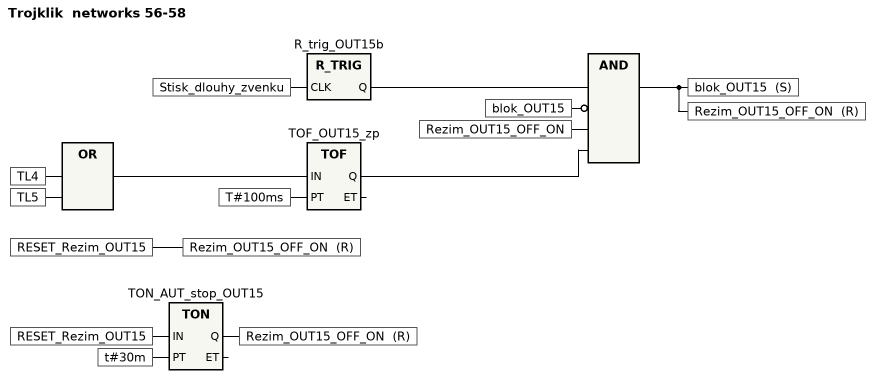
[picture p48: Trojklik (FBD) networks 56-58]
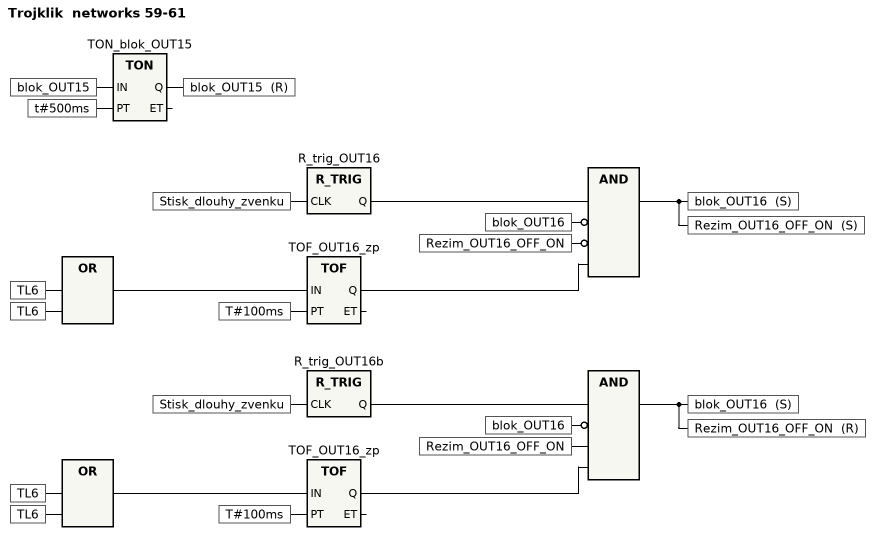
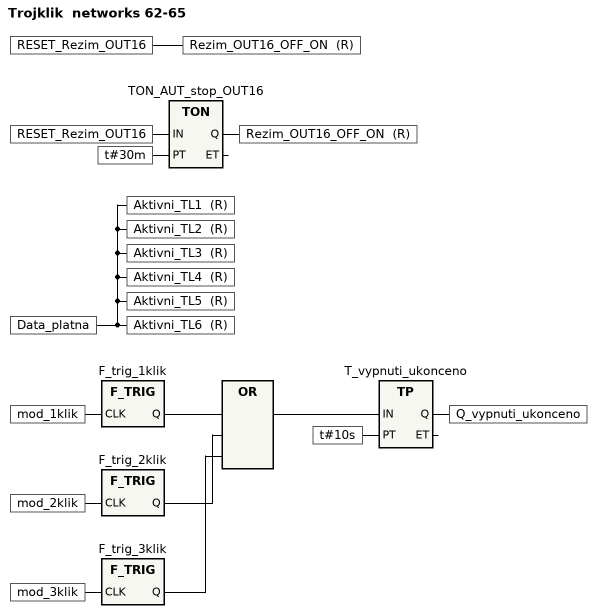
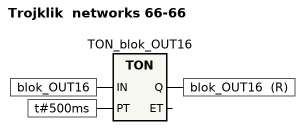
_FBD_ (* Function Block Diagram *)
NETWORK 1
	TP_T_max:TP(IN: T_max:TON(IN: AND(OR(Rezim_1klik_OFF_ON, Rezim_2klik_OFF_ON, Rezim_3klik_OFF_ON), AUT_vyp), PT: cas_vypnuti), PT: t#400ms) => Q_T_MAX
NETWORK 2
	AND(TL1, NOT Aktivni_TL1, NOT Aktivni_TL2, NOT Aktivni_TL3, NOT Aktivni_TL4, NOT Aktivni_TL5, NOT Aktivni_TL6) => S Aktivni_TL1
NETWORK 3
	AND(TL2, NOT Aktivni_TL1, NOT Aktivni_TL2, NOT Aktivni_TL3, NOT Aktivni_TL4, NOT Aktivni_TL5, NOT Aktivni_TL6) => S Aktivni_TL2
NETWORK 4
	AND(TL3, NOT Aktivni_TL1, NOT Aktivni_TL2, NOT Aktivni_TL3, NOT Aktivni_TL4, NOT Aktivni_TL5, NOT Aktivni_TL6) => S Aktivni_TL3
NETWORK 5
	AND(TL4, NOT Aktivni_TL1, NOT Aktivni_TL2, NOT Aktivni_TL3, NOT Aktivni_TL4, NOT Aktivni_TL5, NOT Aktivni_TL6) => S Aktivni_TL4
NETWORK 6
	AND(TL5, NOT Aktivni_TL1, NOT Aktivni_TL2, NOT Aktivni_TL3, NOT Aktivni_TL4, NOT Aktivni_TL5, NOT Aktivni_TL6) => S Aktivni_TL5
NETWORK 7
	AND(TL6, NOT Aktivni_TL1, NOT Aktivni_TL2, NOT Aktivni_TL3, NOT Aktivni_TL4, NOT Aktivni_TL5, NOT Aktivni_TL6) => S Aktivni_TL6
NETWORK 8
	OR(AND(TL1, Aktivni_TL1), AND(TL2, Aktivni_TL2), AND(TL3, Aktivni_TL3)) => TLx_sklad
NETWORK 9
	OR(AND(TL4, Aktivni_TL4), AND(TL5, Aktivni_TL5), AND(TL6, Aktivni_TL6)) => TLx_zvenku
NETWORK 10
	F_trig_hr1:F_TRIG(CLK: TLx_sklad) => TLx_sklad_hr1
NETWORK 11
	F_trig_hr1_zvenku:F_TRIG(CLK: TLx_zvenku) => TLx_sklad_hr1_zvenku
NETWORK 12
	AND(TLx_sklad_hr1, NOT SET_stisk_TLx) => S Stisk_kratky
NETWORK 13
	AND(TLx_sklad_hr1_zvenku, NOT SET_stisk_TLx_zvenku) => S Stisk_kratky_zvenku
NETWORK 14
	TP_byl_kratky:TP(IN: Stisk_kratky, PT: T#4s) => Q_byl_kratky
NETWORK 15
	TP_byl_kratky_zvenku:TP(IN: Stisk_kratky_zvenku, PT: T#4s) => Q_byl_kratky_zvenku
NETWORK 16
	AND(TLx_sklad_hr1, SET_stisk_TLx) => S Stisk_dlouhy
NETWORK 17
	AND(TLx_sklad_hr1_zvenku, SET_stisk_TLx_zvenku) => S Stisk_dlouhy_zvenku
NETWORK 18
	OR(TLx_sklad, TLx_zvenku) => R Stisk_kratky
NETWORK 19
	OR(TLx_zvenku, TLx_sklad) => R Stisk_kratky_zvenku
NETWORK 20
	Stisk_kratky => S blok_kratky
NETWORK 21
	Stisk_kratky_zvenku => S blok_kratky_zvenku
NETWORK 22
	Data_platna => R blok_kratky
NETWORK 23
	Data_platna => R blok_kratky_zvenku
NETWORK 24
	OR(TLx_sklad, TLx_zvenku) => R Stisk_dlouhy
NETWORK 25
	OR(TLx_zvenku, TLx_sklad) => R Stisk_dlouhy_zvenku
NETWORK 26
	AND(NOT mod_1klik, Data_platna, NOT mod_2klik, FALSE, NOT mod_3klik) => R ZAP_VYP_sklad
NETWORK 27
	AND(OR(EQ(TLx_INT, 1), EQ(TLx_INT_zvenku, 1)), NOT mod_1klik, Data_platna, NOT mod_2klik, NOT mod_3klik, NOT ZAP_VYP_sklad, OR(Q_vypnuti_ukonceno, TRUE), NOT blok) => S blok, S mod_1klik
NETWORK 28
	AND(OR(GE(TLx_INT, 1), GE(TLx_INT_zvenku, 1)), OR(Q_vypnuti_ukonceno, TRUE), Data_platna, NOT ZAP_VYP_sklad, NOT blok_ZAP_VYP) => S blok_ZAP_VYP, S ZAP_VYP_sklad
NETWORK 29
	AND(OR(EQ(TLx_INT, 1), EQ(TLx_INT_zvenku, 1)), OR(Data_platna, AND(blok_kratky, TLx_sklad), AND(blok_kratky_zvenku, TLx_zvenku)), ZAP_VYP_sklad, NOT blok_ZAP_VYP, Data_platna, NOT blok_ZAP_VYP, NOT blok) => S blok, R ZAP_VYP_sklad, R mod_1klik
NETWORK 30
	T_blok:TON(IN: blok, PT: T#1s) => R blok
NETWORK 31
	T_blok_ZAP_VYP:TON(IN: blok_ZAP_VYP, PT: T#1s) => R blok_ZAP_VYP
NETWORK 32
	OR(AND(NOT EQ(TLx_INT, 1), NOT EQ(TLx_INT_zvenku, 1), NOT Data_platna, NOT Stisk_dlouhy_zvenku, NOT Stisk_dlouhy, OR(NOT ZAP_VYP_sklad, AND(mod_3klik, FALSE), TRUE, AND(mod_2klik, FALSE)), Data_platna_reset), AND(mod_3klik, FALSE), AND(mod_2klik, FALSE), NOT ZAP_VYP_sklad) => R mod_1klik
NETWORK 33
	AND(OR(EQ(TLx_INT, 2), EQ(TLx_INT_zvenku, 2)), ZAP_VYP_sklad, OR(Q_vypnuti_ukonceno, TRUE), Data_platna) => S mod_2klik
NETWORK 34
	OR(OR(AND(NOT EQ(TLx_INT_zvenku, 2), NOT EQ(TLx_INT, 2), NOT Data_platna, NOT Stisk_dlouhy_zvenku, NOT Stisk_dlouhy, OR(TRUE, NOT ZAP_VYP_sklad, AND(mod_1klik, FALSE), AND(mod_3klik, FALSE)), Data_platna_reset), NOT ZAP_VYP_sklad, AND(mod_3klik, FALSE), AND(mod_1klik, FALSE)), NOT ZAP_VYP_sklad) => R mod_2klik
NETWORK 35
	AND(OR(Q_vypnuti_ukonceno, TRUE), OR(EQ(TLx_INT, 3), EQ(TLx_INT_zvenku, 3)), ZAP_VYP_sklad, Data_platna) => S mod_3klik
NETWORK 36
	OR(OR(AND(NOT EQ(TLx_INT_zvenku, 3), NOT EQ(TLx_INT, 3), NOT Data_platna, NOT Stisk_dlouhy_zvenku, NOT Stisk_dlouhy, OR(TRUE, NOT ZAP_VYP_sklad, AND(mod_1klik, FALSE), AND(mod_2klik, FALSE)), Data_platna_reset), NOT ZAP_VYP_sklad, AND(mod_1klik, FALSE), AND(mod_2klik, FALSE)), NOT ZAP_VYP_sklad) => R mod_3klik
NETWORK 37
	TLx_Citac:CTU(CU: AND(Stisk_kratky, LT(TLx_INT, Pocet_kliku_MAX)), RESET: OR(AND(Data_platna, OR(Q_vypnuti_ukonceno, TRUE)), Q_stisk_TLx), PV: 0, CV => TLx_INT)
NETWORK 38
	TLx_Citac_zvenku:CTU(CU: Stisk_kratky_zvenku, RESET: OR(AND(Data_platna, OR(Q_vypnuti_ukonceno, TRUE)), Q_stisk_TLx_zvenku), PV: 0, CV => TLx_INT_zvenku)
NETWORK 39 (* Data platna *)
	T_Data_platna:TON(IN: AND(NOT TLx_sklad, NOT TLx_zvenku), PT: T#1000ms) => Data_platna
NETWORK 40 (* Data platna *)
	T_Data_platna_reset:TON(IN: AND(NOT TLx_sklad, NOT TLx_zvenku), PT: T#1000ms) => Data_platna_reset
NETWORK 41 (* delka stisku TLx *)
	T_stisk_TLx:TON(IN: AND(TLx_sklad, OR(NOT Q_byl_kratky, TRUE)), PT: T#600ms) => Q_stisk_TLx
NETWORK 42 (* delka stisku TLx *)
	T_stisk_TLx_zvenku:TON(IN: AND(TLx_zvenku, OR(NOT Q_byl_kratky_zvenku, TRUE)), PT: T#600ms) => Q_stisk_TLx_zvenku
NETWORK 43
	SR_stisk_TLx:SR(SET1: Q_stisk_TLx, RESET: R_trig_hr2:R_TRIG(CLK: TLx_sklad)) => SET_stisk_TLx
NETWORK 44
	SR_stisk_TLx_zvenku:SR(SET1: Q_stisk_TLx_zvenku, RESET: R_trig_hr2_zvenku:R_TRIG(CLK: TLx_zvenku)) => SET_stisk_TLx_zvenku
NETWORK 45
	OR(AND(mod_1klik, ZAP_VYP_sklad, TLx_sklad, NOT Q_byl_kratky, mod_1klik, ZAP_VYP_sklad, Q_stisk_TLx), TP_mode_1klik:TP(IN: OR(AND(mod_1klik, ZAP_VYP_sklad, NOT Q_T_MAX, NOT RESET_Rezim_1klik, NOT Q_vypnuti_ukonceno, Data_platna, OR(Stisk_kratky, Stisk_kratky_zvenku)), AND(NOT ZAP_VYP_sklad, OR(Stisk_kratky, Stisk_kratky_zvenku), NOT Q_T_MAX, NOT RESET_Rezim_1klik, FALSE, mod_1klik)), PT: t#400ms), tp_1klik_vyp:TP(IN: AND(f_trig_1klik_vyp:F_TRIG(CLK: mod_1klik), NOT RESET_Rezim_1klik, NOT Q_T_MAX), PT: t#400ms), TP_reset1:TP(IN: AND(mod_1klik, ZAP_VYP_sklad, OR(RESET_Rezim_1klik, Q_T_MAX)), PT: t#400ms)) => Rezim_1klik_PULS
NETWORK 46
	AND(ZAP_VYP_sklad, mod_1klik) => Rezim_1klik_OFF_ON
NETWORK 47
	OR(AND(mod_2klik, ZAP_VYP_sklad, NOT Q_byl_kratky, mod_2klik, ZAP_VYP_sklad, TLx_sklad, Q_stisk_TLx), TP_mode_2klik:TP(IN: OR(AND(mod_2klik, ZAP_VYP_sklad, NOT Q_T_MAX, NOT RESET_Rezim_2klik, NOT Q_vypnuti_ukonceno, Data_platna, OR(Stisk_kratky, Stisk_kratky_zvenku)), AND(NOT ZAP_VYP_sklad, NOT Q_T_MAX, NOT RESET_Rezim_2klik, FALSE, OR(Stisk_kratky, Stisk_kratky_zvenku), mod_2klik)), PT: t#400ms), tp_2klik_vyp:TP(IN: AND(f_trig_2klik_vyp:F_TRIG(CLK: mod_2klik), NOT RESET_Rezim_2klik, NOT Q_T_MAX), PT: t#400ms), TP_reset2:TP(IN: AND(mod_2klik, ZAP_VYP_sklad, OR(RESET_Rezim_2klik, Q_T_MAX)), PT: t#400ms)) => Rezim_2klik_PULS
NETWORK 48
	AND(ZAP_VYP_sklad, mod_2klik) => Rezim_2klik_OFF_ON
NETWORK 49
	OR(AND(mod_3klik, ZAP_VYP_sklad, NOT Q_byl_kratky, mod_3klik, ZAP_VYP_sklad, TLx_sklad, Q_stisk_TLx), TP_mode_3klik:TP(IN: OR(AND(mod_3klik, NOT Q_T_MAX, NOT RESET_Rezim_3klik, NOT Q_vypnuti_ukonceno, Data_platna, ZAP_VYP_sklad, OR(Stisk_kratky, Stisk_kratky_zvenku)), AND(NOT ZAP_VYP_sklad, NOT Q_T_MAX, NOT RESET_Rezim_3klik, FALSE, OR(Stisk_kratky, Stisk_kratky_zvenku), mod_3klik)), PT: t#400ms), tp_3klik_vyp:TP(IN: AND(f_trig_3klik_vyp:F_TRIG(CLK: mod_3klik), NOT RESET_Rezim_3klik, NOT Q_T_MAX), PT: t#400ms), TP_reset3:TP(IN: AND(mod_3klik, ZAP_VYP_sklad, OR(RESET_Rezim_3klik, Q_T_MAX)), PT: t#400ms)) => Rezim_3klik_PULS
NETWORK 50
	AND(ZAP_VYP_sklad, mod_3klik) => Rezim_3klik_OFF_ON
NETWORK 51
	OR(AND(mod_1klik, RESET_Rezim_1klik), AND(mod_2klik, RESET_Rezim_2klik), AND(mod_3klik, RESET_Rezim_3klik), Q_T_MAX) => R ZAP_VYP_sklad
NETWORK 52
	OR(AND(mod_1klik, RESET_Rezim_1klik), Q_T_MAX) => R mod_1klik
NETWORK 53
	OR(AND(mod_2klik, RESET_Rezim_2klik), Q_T_MAX) => R mod_2klik
NETWORK 54
	OR(AND(mod_3klik, RESET_Rezim_3klik), Q_T_MAX) => R mod_3klik
NETWORK 55
	AND(R_trig_OUT15:R_TRIG(CLK: Stisk_dlouhy_zvenku), NOT blok_OUT15, NOT Rezim_OUT15_OFF_ON, TOF_OUT15_zp:TOF(IN: OR(TL4, TL5), PT: T#100ms)) => S blok_OUT15, S Rezim_OUT15_OFF_ON
NETWORK 56
	AND(R_trig_OUT15b:R_TRIG(CLK: Stisk_dlouhy_zvenku), NOT blok_OUT15, Rezim_OUT15_OFF_ON, TOF_OUT15_zp:TOF(IN: OR(TL4, TL5), PT: T#100ms)) => S blok_OUT15, R Rezim_OUT15_OFF_ON
NETWORK 57
	RESET_Rezim_OUT15 => R Rezim_OUT15_OFF_ON
NETWORK 58
	TON_AUT_stop_OUT15:TON(IN: RESET_Rezim_OUT15, PT: t#30m) => R Rezim_OUT15_OFF_ON
NETWORK 59
	TON_blok_OUT15:TON(IN: blok_OUT15, PT: t#500ms) => R blok_OUT15
NETWORK 60
	AND(R_trig_OUT16:R_TRIG(CLK: Stisk_dlouhy_zvenku), NOT blok_OUT16, NOT Rezim_OUT16_OFF_ON, TOF_OUT16_zp:TOF(IN: OR(TL6, TL6), PT: T#100ms)) => S blok_OUT16, S Rezim_OUT16_OFF_ON
NETWORK 61
	AND(R_trig_OUT16b:R_TRIG(CLK: Stisk_dlouhy_zvenku), NOT blok_OUT16, Rezim_OUT16_OFF_ON, TOF_OUT16_zp:TOF(IN: OR(TL6, TL6), PT: T#100ms)) => S blok_OUT16, R Rezim_OUT16_OFF_ON
NETWORK 62
	RESET_Rezim_OUT16 => R Rezim_OUT16_OFF_ON
NETWORK 63
	TON_AUT_stop_OUT16:TON(IN: RESET_Rezim_OUT16, PT: t#30m) => R Rezim_OUT16_OFF_ON
NETWORK 64
	Data_platna => R Aktivni_TL1, R Aktivni_TL2, R Aktivni_TL3, R Aktivni_TL4, R Aktivni_TL5, R Aktivni_TL6
NETWORK 65
	T_vypnuti_ukonceno:TP(IN: OR(F_trig_1klik:F_TRIG(CLK: mod_1klik), F_trig_2klik:F_TRIG(CLK: mod_2klik), F_trig_3klik:F_TRIG(CLK: mod_3klik)), PT: t#10s) => Q_vypnuti_ukonceno
NETWORK 66
	TON_blok_OUT16:TON(IN: blok_OUT16, PT: t#500ms) => R blok_OUT16
_END_FBD_
(* the same logic as Structured Text *)
(* Network 1 *)
T_max(IN := (Rezim_1klik_OFF_ON OR Rezim_2klik_OFF_ON OR Rezim_3klik_OFF_ON) AND AUT_vyp, PT := cas_vypnuti);
TP_T_max(IN := T_max.Q, PT := t#400ms);
Q_T_MAX := TP_T_max.Q;
(* Network 2 *)
IF TL1 AND NOT Aktivni_TL1 AND NOT Aktivni_TL2 AND NOT Aktivni_TL3 AND NOT Aktivni_TL4 AND NOT Aktivni_TL5 AND NOT Aktivni_TL6 THEN Aktivni_TL1 := TRUE; END_IF;
(* Network 3 *)
IF TL2 AND NOT Aktivni_TL1 AND NOT Aktivni_TL2 AND NOT Aktivni_TL3 AND NOT Aktivni_TL4 AND NOT Aktivni_TL5 AND NOT Aktivni_TL6 THEN Aktivni_TL2 := TRUE; END_IF;
(* Network 4 *)
IF TL3 AND NOT Aktivni_TL1 AND NOT Aktivni_TL2 AND NOT Aktivni_TL3 AND NOT Aktivni_TL4 AND NOT Aktivni_TL5 AND NOT Aktivni_TL6 THEN Aktivni_TL3 := TRUE; END_IF;
(* Network 5 *)
IF TL4 AND NOT Aktivni_TL1 AND NOT Aktivni_TL2 AND NOT Aktivni_TL3 AND NOT Aktivni_TL4 AND NOT Aktivni_TL5 AND NOT Aktivni_TL6 THEN Aktivni_TL4 := TRUE; END_IF;
(* Network 6 *)
IF TL5 AND NOT Aktivni_TL1 AND NOT Aktivni_TL2 AND NOT Aktivni_TL3 AND NOT Aktivni_TL4 AND NOT Aktivni_TL5 AND NOT Aktivni_TL6 THEN Aktivni_TL5 := TRUE; END_IF;
(* Network 7 *)
IF TL6 AND NOT Aktivni_TL1 AND NOT Aktivni_TL2 AND NOT Aktivni_TL3 AND NOT Aktivni_TL4 AND NOT Aktivni_TL5 AND NOT Aktivni_TL6 THEN Aktivni_TL6 := TRUE; END_IF;
(* Network 8 *)
TLx_sklad := (TL1 AND Aktivni_TL1) OR (TL2 AND Aktivni_TL2) OR (TL3 AND Aktivni_TL3);
(* Network 9 *)
TLx_zvenku := (TL4 AND Aktivni_TL4) OR (TL5 AND Aktivni_TL5) OR (TL6 AND Aktivni_TL6);
(* Network 10 *)
F_trig_hr1(CLK := TLx_sklad);
TLx_sklad_hr1 := F_trig_hr1.Q;
(* Network 11 *)
F_trig_hr1_zvenku(CLK := TLx_zvenku);
TLx_sklad_hr1_zvenku := F_trig_hr1_zvenku.Q;
(* Network 12 *)
IF TLx_sklad_hr1 AND NOT SET_stisk_TLx THEN Stisk_kratky := TRUE; END_IF;
(* Network 13 *)
IF TLx_sklad_hr1_zvenku AND NOT SET_stisk_TLx_zvenku THEN Stisk_kratky_zvenku := TRUE; END_IF;
(* Network 14 *)
TP_byl_kratky(IN := Stisk_kratky, PT := T#4s);
Q_byl_kratky := TP_byl_kratky.Q;
(* Network 15 *)
TP_byl_kratky_zvenku(IN := Stisk_kratky_zvenku, PT := T#4s);
Q_byl_kratky_zvenku := TP_byl_kratky_zvenku.Q;
(* Network 16 *)
IF TLx_sklad_hr1 AND SET_stisk_TLx THEN Stisk_dlouhy := TRUE; END_IF;
(* Network 17 *)
IF TLx_sklad_hr1_zvenku AND SET_stisk_TLx_zvenku THEN Stisk_dlouhy_zvenku := TRUE; END_IF;
(* Network 18 *)
IF TLx_sklad OR TLx_zvenku THEN Stisk_kratky := FALSE; END_IF;
(* Network 19 *)
IF TLx_zvenku OR TLx_sklad THEN Stisk_kratky_zvenku := FALSE; END_IF;
(* Network 20 *)
IF Stisk_kratky THEN blok_kratky := TRUE; END_IF;
(* Network 21 *)
IF Stisk_kratky_zvenku THEN blok_kratky_zvenku := TRUE; END_IF;
(* Network 22 *)
IF Data_platna THEN blok_kratky := FALSE; END_IF;
(* Network 23 *)
IF Data_platna THEN blok_kratky_zvenku := FALSE; END_IF;
(* Network 24 *)
IF TLx_sklad OR TLx_zvenku THEN Stisk_dlouhy := FALSE; END_IF;
(* Network 25 *)
IF TLx_zvenku OR TLx_sklad THEN Stisk_dlouhy_zvenku := FALSE; END_IF;
(* Network 26 *)
IF NOT mod_1klik AND Data_platna AND NOT mod_2klik AND FALSE AND NOT mod_3klik THEN ZAP_VYP_sklad := FALSE; END_IF;
(* Network 27 *)
_p1 := ((TLx_INT = 1) OR (TLx_INT_zvenku = 1)) AND NOT mod_1klik AND Data_platna AND NOT mod_2klik AND NOT mod_3klik AND NOT ZAP_VYP_sklad AND (Q_vypnuti_ukonceno OR TRUE) AND NOT blok;
IF _p1 THEN blok := TRUE; mod_1klik := TRUE; END_IF;
(* Network 28 *)
_p2 := ((TLx_INT >= 1) OR (TLx_INT_zvenku >= 1)) AND (Q_vypnuti_ukonceno OR TRUE) AND Data_platna AND NOT ZAP_VYP_sklad AND NOT blok_ZAP_VYP;
IF _p2 THEN blok_ZAP_VYP := TRUE; ZAP_VYP_sklad := TRUE; END_IF;
(* Network 29 *)
_p3 := ((TLx_INT = 1) OR (TLx_INT_zvenku = 1)) AND (Data_platna OR (blok_kratky AND TLx_sklad) OR (blok_kratky_zvenku AND TLx_zvenku)) AND ZAP_VYP_sklad AND NOT blok_ZAP_VYP AND Data_platna AND NOT blok_ZAP_VYP AND NOT blok;
IF _p3 THEN blok := TRUE; ZAP_VYP_sklad := FALSE; mod_1klik := FALSE; END_IF;
(* Network 30 *)
T_blok(IN := blok, PT := T#1s);
IF T_blok.Q THEN blok := FALSE; END_IF;
(* Network 31 *)
T_blok_ZAP_VYP(IN := blok_ZAP_VYP, PT := T#1s);
IF T_blok_ZAP_VYP.Q THEN blok_ZAP_VYP := FALSE; END_IF;
(* Network 32 *)
IF (NOT (TLx_INT = 1) AND NOT (TLx_INT_zvenku = 1) AND NOT Data_platna AND NOT Stisk_dlouhy_zvenku AND NOT Stisk_dlouhy AND (NOT ZAP_VYP_sklad OR (mod_3klik AND FALSE) OR TRUE OR (mod_2klik AND FALSE)) AND Data_platna_reset) OR (mod_3klik AND FALSE) OR (mod_2klik AND FALSE) OR NOT ZAP_VYP_sklad THEN mod_1klik := FALSE; END_IF;
(* Network 33 *)
IF ((TLx_INT = 2) OR (TLx_INT_zvenku = 2)) AND ZAP_VYP_sklad AND (Q_vypnuti_ukonceno OR TRUE) AND Data_platna THEN mod_2klik := TRUE; END_IF;
(* Network 34 *)
IF ((NOT (TLx_INT_zvenku = 2) AND NOT (TLx_INT = 2) AND NOT Data_platna AND NOT Stisk_dlouhy_zvenku AND NOT Stisk_dlouhy AND (TRUE OR NOT ZAP_VYP_sklad OR (mod_1klik AND FALSE) OR (mod_3klik AND FALSE)) AND Data_platna_reset) OR NOT ZAP_VYP_sklad OR (mod_3klik AND FALSE) OR (mod_1klik AND FALSE)) OR NOT ZAP_VYP_sklad THEN mod_2klik := FALSE; END_IF;
(* Network 35 *)
IF (Q_vypnuti_ukonceno OR TRUE) AND ((TLx_INT = 3) OR (TLx_INT_zvenku = 3)) AND ZAP_VYP_sklad AND Data_platna THEN mod_3klik := TRUE; END_IF;
(* Network 36 *)
IF ((NOT (TLx_INT_zvenku = 3) AND NOT (TLx_INT = 3) AND NOT Data_platna AND NOT Stisk_dlouhy_zvenku AND NOT Stisk_dlouhy AND (TRUE OR NOT ZAP_VYP_sklad OR (mod_1klik AND FALSE) OR (mod_2klik AND FALSE)) AND Data_platna_reset) OR NOT ZAP_VYP_sklad OR (mod_1klik AND FALSE) OR (mod_2klik AND FALSE)) OR NOT ZAP_VYP_sklad THEN mod_3klik := FALSE; END_IF;
(* Network 37 *)
TLx_Citac(CU := Stisk_kratky AND (TLx_INT < Pocet_kliku_MAX), RESET := (Data_platna AND (Q_vypnuti_ukonceno OR TRUE)) OR Q_stisk_TLx, PV := 0);
TLx_INT := TLx_Citac.CV;
(* Network 38 *)
TLx_Citac_zvenku(CU := Stisk_kratky_zvenku, RESET := (Data_platna AND (Q_vypnuti_ukonceno OR TRUE)) OR Q_stisk_TLx_zvenku, PV := 0);
TLx_INT_zvenku := TLx_Citac_zvenku.CV;
(* Network 39 *)
T_Data_platna(IN := NOT TLx_sklad AND NOT TLx_zvenku, PT := T#1000ms);
Data_platna := T_Data_platna.Q;
(* Network 40 *)
T_Data_platna_reset(IN := NOT TLx_sklad AND NOT TLx_zvenku, PT := T#1000ms);
Data_platna_reset := T_Data_platna_reset.Q;
(* Network 41: see the listing above *)
(* Network 42: see the listing above *)
(* Network 43 *)
R_trig_hr2(CLK := TLx_sklad);
SR_stisk_TLx(SET1 := Q_stisk_TLx, RESET := R_trig_hr2.Q);
SET_stisk_TLx := SR_stisk_TLx.Q1;
(* Network 44 *)
R_trig_hr2_zvenku(CLK := TLx_zvenku);
SR_stisk_TLx_zvenku(SET1 := Q_stisk_TLx_zvenku, RESET := R_trig_hr2_zvenku.Q);
SET_stisk_TLx_zvenku := SR_stisk_TLx_zvenku.Q1;
(* Network 45 *)
TP_mode_1klik(IN := (mod_1klik AND ZAP_VYP_sklad AND NOT Q_T_MAX AND NOT RESET_Rezim_1klik AND NOT Q_vypnuti_ukonceno AND Data_platna AND (Stisk_kratky OR Stisk_kratky_zvenku)) OR (NOT ZAP_VYP_sklad AND (Stisk_kratky OR Stisk_kratky_zvenku) AND NOT Q_T_MAX AND NOT RESET_Rezim_1klik AND FALSE AND mod_1klik), PT := t#400ms);
f_trig_1klik_vyp(CLK := mod_1klik);
tp_1klik_vyp(IN := f_trig_1klik_vyp.Q AND NOT RESET_Rezim_1klik AND NOT Q_T_MAX, PT := t#400ms);
TP_reset1(IN := mod_1klik AND ZAP_VYP_sklad AND (RESET_Rezim_1klik OR Q_T_MAX), PT := t#400ms);
Rezim_1klik_PULS := (mod_1klik AND ZAP_VYP_sklad AND TLx_sklad AND NOT Q_byl_kratky AND mod_1klik AND ZAP_VYP_sklad AND Q_stisk_TLx) OR TP_mode_1klik.Q OR tp_1klik_vyp.Q OR TP_reset1.Q;
(* Network 46 *)
Rezim_1klik_OFF_ON := ZAP_VYP_sklad AND mod_1klik;
(* Network 47 *)
TP_mode_2klik(IN := (mod_2klik AND ZAP_VYP_sklad AND NOT Q_T_MAX AND NOT RESET_Rezim_2klik AND NOT Q_vypnuti_ukonceno AND Data_platna AND (Stisk_kratky OR Stisk_kratky_zvenku)) OR (NOT ZAP_VYP_sklad AND NOT Q_T_MAX AND NOT RESET_Rezim_2klik AND FALSE AND (Stisk_kratky OR Stisk_kratky_zvenku) AND mod_2klik), PT := t#400ms);
f_trig_2klik_vyp(CLK := mod_2klik);
tp_2klik_vyp(IN := f_trig_2klik_vyp.Q AND NOT RESET_Rezim_2klik AND NOT Q_T_MAX, PT := t#400ms);
TP_reset2(IN := mod_2klik AND ZAP_VYP_sklad AND (RESET_Rezim_2klik OR Q_T_MAX), PT := t#400ms);
Rezim_2klik_PULS := (mod_2klik AND ZAP_VYP_sklad AND NOT Q_byl_kratky AND mod_2klik AND ZAP_VYP_sklad AND TLx_sklad AND Q_stisk_TLx) OR TP_mode_2klik.Q OR tp_2klik_vyp.Q OR TP_reset2.Q;
(* Network 48 *)
Rezim_2klik_OFF_ON := ZAP_VYP_sklad AND mod_2klik;
(* Network 49 *)
TP_mode_3klik(IN := (mod_3klik AND NOT Q_T_MAX AND NOT RESET_Rezim_3klik AND NOT Q_vypnuti_ukonceno AND Data_platna AND ZAP_VYP_sklad AND (Stisk_kratky OR Stisk_kratky_zvenku)) OR (NOT ZAP_VYP_sklad AND NOT Q_T_MAX AND NOT RESET_Rezim_3klik AND FALSE AND (Stisk_kratky OR Stisk_kratky_zvenku) AND mod_3klik), PT := t#400ms);
f_trig_3klik_vyp(CLK := mod_3klik);
tp_3klik_vyp(IN := f_trig_3klik_vyp.Q AND NOT RESET_Rezim_3klik AND NOT Q_T_MAX, PT := t#400ms);
TP_reset3(IN := mod_3klik AND ZAP_VYP_sklad AND (RESET_Rezim_3klik OR Q_T_MAX), PT := t#400ms);
Rezim_3klik_PULS := (mod_3klik AND ZAP_VYP_sklad AND NOT Q_byl_kratky AND mod_3klik AND ZAP_VYP_sklad AND TLx_sklad AND Q_stisk_TLx) OR TP_mode_3klik.Q OR tp_3klik_vyp.Q OR TP_reset3.Q;
(* Network 50 *)
Rezim_3klik_OFF_ON := ZAP_VYP_sklad AND mod_3klik;
(* Network 51 *)
IF (mod_1klik AND RESET_Rezim_1klik) OR (mod_2klik AND RESET_Rezim_2klik) OR (mod_3klik AND RESET_Rezim_3klik) OR Q_T_MAX THEN ZAP_VYP_sklad := FALSE; END_IF;
(* Network 52 *)
IF (mod_1klik AND RESET_Rezim_1klik) OR Q_T_MAX THEN mod_1klik := FALSE; END_IF;
(* Network 53 *)
IF (mod_2klik AND RESET_Rezim_2klik) OR Q_T_MAX THEN mod_2klik := FALSE; END_IF;
(* Network 54 *)
IF (mod_3klik AND RESET_Rezim_3klik) OR Q_T_MAX THEN mod_3klik := FALSE; END_IF;
(* Network 55 *)
R_trig_OUT15(CLK := Stisk_dlouhy_zvenku);
TOF_OUT15_zp(IN := TL4 OR TL5, PT := T#100ms);
_p4 := R_trig_OUT15.Q AND NOT blok_OUT15 AND NOT Rezim_OUT15_OFF_ON AND TOF_OUT15_zp.Q;
IF _p4 THEN blok_OUT15 := TRUE; Rezim_OUT15_OFF_ON := TRUE; END_IF;
(* Network 56 *)
R_trig_OUT15b(CLK := Stisk_dlouhy_zvenku);
TOF_OUT15_zp(IN := TL4 OR TL5, PT := T#100ms);
_p5 := R_trig_OUT15b.Q AND NOT blok_OUT15 AND Rezim_OUT15_OFF_ON AND TOF_OUT15_zp.Q;
IF _p5 THEN blok_OUT15 := TRUE; Rezim_OUT15_OFF_ON := FALSE; END_IF;
(* Network 57 *)
IF RESET_Rezim_OUT15 THEN Rezim_OUT15_OFF_ON := FALSE; END_IF;
(* Network 58 *)
TON_AUT_stop_OUT15(IN := RESET_Rezim_OUT15, PT := t#30m);
IF TON_AUT_stop_OUT15.Q THEN Rezim_OUT15_OFF_ON := FALSE; END_IF;
(* Network 59 *)
TON_blok_OUT15(IN := blok_OUT15, PT := t#500ms);
IF TON_blok_OUT15.Q THEN blok_OUT15 := FALSE; END_IF;
(* Network 60 *)
R_trig_OUT16(CLK := Stisk_dlouhy_zvenku);
TOF_OUT16_zp(IN := TL6 OR TL6, PT := T#100ms);
_p6 := R_trig_OUT16.Q AND NOT blok_OUT16 AND NOT Rezim_OUT16_OFF_ON AND TOF_OUT16_zp.Q;
IF _p6 THEN blok_OUT16 := TRUE; Rezim_OUT16_OFF_ON := TRUE; END_IF;
(* Network 61 *)
R_trig_OUT16b(CLK := Stisk_dlouhy_zvenku);
TOF_OUT16_zp(IN := TL6 OR TL6, PT := T#100ms);
_p7 := R_trig_OUT16b.Q AND NOT blok_OUT16 AND Rezim_OUT16_OFF_ON AND TOF_OUT16_zp.Q;
IF _p7 THEN blok_OUT16 := TRUE; Rezim_OUT16_OFF_ON := FALSE; END_IF;
(* Network 62 *)
IF RESET_Rezim_OUT16 THEN Rezim_OUT16_OFF_ON := FALSE; END_IF;
(* Network 63 *)
TON_AUT_stop_OUT16(IN := RESET_Rezim_OUT16, PT := t#30m);
IF TON_AUT_stop_OUT16.Q THEN Rezim_OUT16_OFF_ON := FALSE; END_IF;
(* Network 64 *)
IF Data_platna THEN Aktivni_TL1 := FALSE; Aktivni_TL2 := FALSE; Aktivni_TL3 := FALSE; Aktivni_TL4 := FALSE; Aktivni_TL5 := FALSE; Aktivni_TL6 := FALSE; END_IF;
(* Network 65 *)
F_trig_1klik(CLK := mod_1klik);
F_trig_2klik(CLK := mod_2klik);
F_trig_3klik(CLK := mod_3klik);
T_vypnuti_ukonceno(IN := F_trig_1klik.Q OR F_trig_2klik.Q OR F_trig_3klik.Q, PT := t#10s);
Q_vypnuti_ukonceno := T_vypnuti_ukonceno.Q;
(* Network 66 *)
TON_blok_OUT16(IN := blok_OUT16, PT := t#500ms);
IF TON_blok_OUT16.Q THEN blok_OUT16 := FALSE; END_IF;
END_FUNCTION_BLOCK

(* POU Zhasni, ST *)
FUNCTION_BLOCK Zhasni
VAR_INPUT
	wIn: WORD;
	xPresun: BOOL;
END_VAR
VAR_OUTPUT
	xonOUT1: BOOL;
	xonOUT2: BOOL;
	xonOUT3: BOOL;

	xoffOUT1: BOOL;
	xoffOUT2: BOOL;
	xoffOUT3: BOOL;
	wLast: WORD;
	xPresunuto: BOOL;
END_VAR
VAR
	start: BOOL;
	TP1: TP;
	stav: WORD;
	last: WORD;
	F_TRIG5: F_TRIG;
END_VAR
IF xPresun=TRUE THEN
	stav:=wIn;
	start:=TRUE;


CASE stav OF
	2: 	xonOUT2:=TRUE;
		last:=2;
	3: 	xonOUT3:=TRUE;
		last:=3;
END_CASE


IF wLast=0 AND stav=1 THEN
xonOUT1:=TRUE;
last:=1;
END_IF

IF NOT( wLast=0) AND stav=1 THEN
	CASE wLast OF
	1: xoffOUT1:=TRUE;
		last:=0;
	2: xoffOUT2:=TRUE;
		last:=0;
	3: xoffOUT3:=TRUE;
		last:=0;
	END_CASE

END_IF
END_IF

TP1(IN:=start , PT:=t#50ms , Q=> , ET=> );
F_TRIG5(CLK:=TP1.Q , Q=> );
IF F_TRIG5.Q=TRUE THEN
	wLast:=last;
	start:=FALSE;
	xoffOUT1:=FALSE;
	xoffOUT2:=FALSE;
	xoffOUT3:=FALSE;
	xonOUT1:=FALSE;
	xonOUT2:=FALSE;
	xonOUT3:=FALSE;
END_IF

xPresunuto:=xPresun;
END_FUNCTION_BLOCK

(* POU dali/Ovladani_7_8_9, ST *)
FUNCTION_BLOCK Ovladani_7_8_9
VAR_INPUT
	xVstup: BOOL;
	rCidlo: REAL;
	rUroven1: REAL;
	rUroven2: REAL;
	tZpozdeniCidla: TIME;
END_VAR
VAR_OUTPUT
	On_7: BOOL;
	On_8: BOOL;
	On_9: BOOL;
	Off_7: BOOL;
	Off_8: BOOL;
	Off_9: BOOL;
END_VAR
VAR
	Stav7: BOOL;
	Stav8: BOOL;
	Stav9: BOOL;
	StavSvetel: BOOL;
	Zmacknuto: BOOL;
	R_TRIG1: R_TRIG;
	F_TRIG1: F_TRIG;
	BLINK1: BLINK;

END_VAR
R_TRIG1(CLK:=xVstup, Q=>Zmacknuto );
F_TRIG1(CLK:=xVstup);
BLINK1(ENABLE:=TRUE , TIMELOW:=tZpozdeniCidla , TIMEHIGH:=t#1s);

IF BLINK1.OUT THEN Cidlo_zpozdene:=rCidlo;
END_IF

StavSvetel:=Stav7 OR Stav8 OR Stav9;

IF Zmacknuto AND (StavSvetel=FALSE) THEN		(*vse zhasnuto*)
	On_7:=TRUE;
	On_8:=TRUE;
	On_9:=TRUE;
	Stav7:=TRUE;
	Stav8:=TRUE;
	Stav9:=TRUE;
END_IF

IF Zmacknuto AND (StavSvetel=TRUE) THEN		(*neco rozsviceno*)
	Off_7:=TRUE;
	Off_8:=TRUE;
	Off_9:=TRUE;
	Stav7:=FALSE;
	Stav8:=FALSE;
	Stav9:=FALSE;
END_IF

IF F_TRIG1.Q THEN
	On_7:=FALSE;
	On_8:=FALSE;
	On_9:=FALSE;
	Off_7:=FALSE;
	Off_8:=FALSE;
	Off_9:=FALSE;
END_IF

IF Cidlo_zpozdene>rUroven1 THEN
	On_7:=FALSE;
	Off_7:=TRUE;
	Stav7:=FALSE;
ELSIF StavSvetel THEN
	On_7:=TRUE;
	Off_7:=FALSE;
	Stav7:=TRUE;
END_IF

IF Cidlo_zpozdene>rUroven2 THEN
	On_9:=FALSE;
	Off_9:=TRUE;
	Stav9:=FALSE;
ELSIF StavSvetel THEN
	On_9:=TRUE;
	Off_9:=FALSE;
	Stav9:=TRUE;
END_IF

IF Zmacknuto AND (StavSvetel=TRUE) THEN		(*neco rozsviceno*)
	Off_7:=TRUE;
	Off_8:=TRUE;
	Off_9:=TRUE;
	Stav7:=FALSE;
	Stav8:=FALSE;
	Stav9:=FALSE;
END_IF

IF F_TRIG1.Q THEN
	On_7:=FALSE;
	On_8:=FALSE;
	On_9:=FALSE;
	Off_7:=FALSE;
	Off_8:=FALSE;
	Off_9:=FALSE;
END_IF
END_FUNCTION_BLOCK

(* POU TriFaze, ST *)
PROGRAM TriFaze
VAR

	Fb750_493_Master3Phase1: Fb750_493_Master3Phase;
	abIn AT %IB22: ARRAY [0..11] OF BYTE;
	abOut AT %QB6: ARRAY [0..11] OF BYTE;

	typ3faze: typConfig3Phase;
	awProud: ARRAY [1..3] OF WORD;
	awNapeti: ARRAY [1..3] OF WORD;
	aiCosFi: ARRAY [1..3] OF INT;
	aiVykon: ARRAY [1..3] OF INT;
	adwSpotreba: ARRAY [1..3] OF DWORD;

	arProud: ARRAY [1..3] OF REAL;
	arNapeti: ARRAY [1..3] OF REAL;
	arCosFi: ARRAY [1..3] OF REAL;
	arVykon: ARRAY [1..3] OF REAL;
	arSpotreba: ARRAY [1..3] OF REAL;
	SmazL1: BOOL;
	SmazL2: BOOL;
	SmazL3: BOOL;
END_VAR
Fb750_493_Master3Phase1(
	xEnable:= TRUE,
	tCycleTime:= ,
	x750_493_000_001:=FALSE ,
	xSaveEnergyConsumption:= ,
	xDeleteEnergyConsumptionL1:=SmazL1 ,
	xDeleteEnergyConsumptionL2:=SmazL1 ,
	xDeleteEnergyConsumptionL3:=SmazL1 ,
	abIn_Data_750_493:=abIn ,
	abOut_Data_750_493:=abOut ,
	typConfig3Phase:=typ3faze ,
	xReady=> ,
	abError=> , 
	awCurrent=>awProud ,
	awVoltage=>awNapeti ,
	aiPowerFactor=>aiCosFi ,
	aiEffectivePower=>aiVykon ,
	adwEnergyConsumption=>adwSpotreba ,
	awMaxCurrent=> , 
	awMaxVoltage=> , 
	awMinCurrent=> ,
	awMinVoltage=> );

arProud[1]:=awProud[1]/1000.0;
arProud[2]:=awProud[2]/1000.0;
arProud[3]:=awProud[3]/1000.0;

arNapeti[1]:=awNapeti[1]/10.0;
arNapeti[2]:=awNapeti[2]/10.0;
arNapeti[3]:=awNapeti[3]/10.0;

arCosFi[1]:=aiCosFi[1]/100.0;
arCosFi[2]:=aiCosFi[2]/100.0;
arCosFi[3]:=aiCosFi[3]/100.0;

arVykon[1]:=aiVykon[1]/10000.0;
arVykon[2]:=aiVykon[2]/10000.0;
arVykon[3]:=aiVykon[3]/10000.0;
;
END_PROGRAM

(* POU PrirazeniVzdalenychPromenych, CFC *)
PROGRAM PrirazeniVzdalenychPromenych
VAR
	d1: D_klop;
	d2: D_klop;
	d3: D_klop;
	d4: D_klop;
	d5: D_klop;
	d6: D_klop;
	d7: D_klop;
	d8: D_klop;
END_VAR
VAR (* helpers for the ST form of the networks *)
	_t91 : REAL;
END_VAR
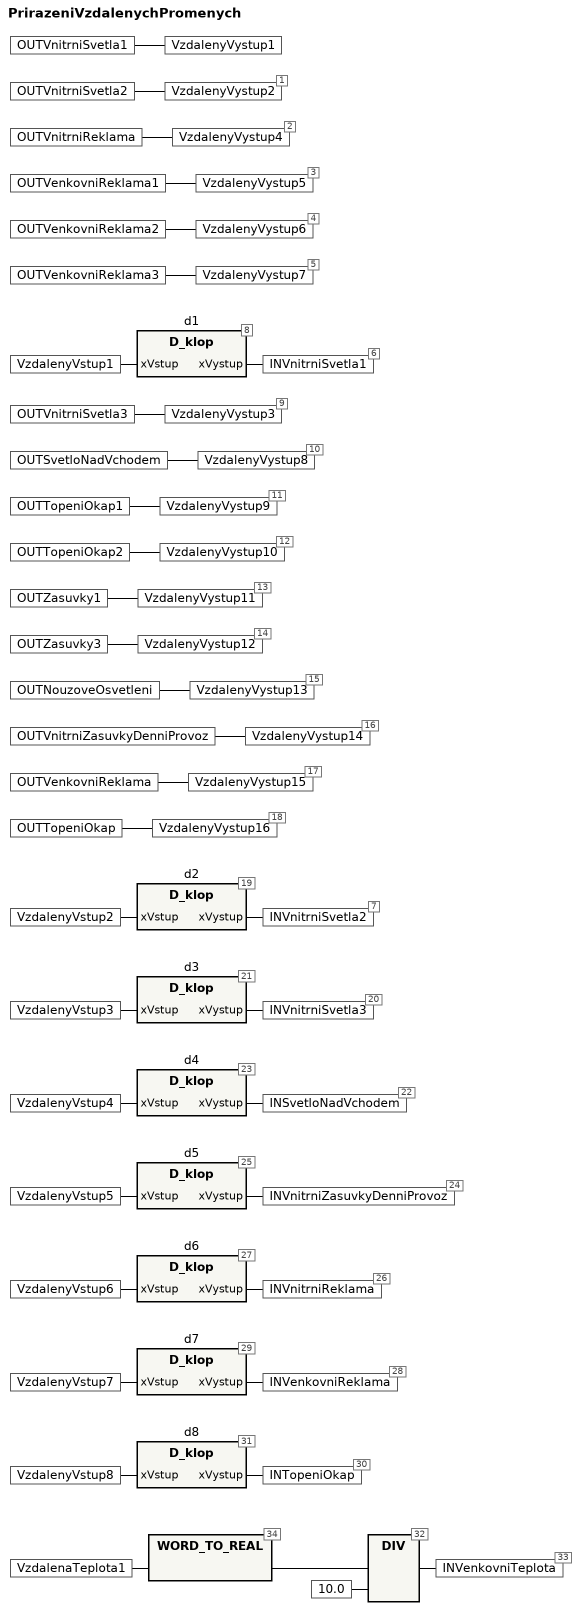
_CFC_ (* Continuous Function Chart, elements in execution order *)
#0 VzdalenyVystup1 <= OUTVnitrniSvetla1
#1 VzdalenyVystup2 <= OUTVnitrniSvetla2
#2 VzdalenyVystup4 <= OUTVnitrniReklama
#3 VzdalenyVystup5 <= OUTVenkovniReklama1
#4 VzdalenyVystup6 <= OUTVenkovniReklama2
#5 VzdalenyVystup7 <= OUTVenkovniReklama3
#6 INVnitrniSvetla1 <= #8.xVystup
#7 INVnitrniSvetla2 <= #19.xVystup
#8 d1:D_klop(xVstup: VzdalenyVstup1)
#9 VzdalenyVystup3 <= OUTVnitrniSvetla3
#10 VzdalenyVystup8 <= OUTSvetloNadVchodem
#11 VzdalenyVystup9 <= OUTTopeniOkap1
#12 VzdalenyVystup10 <= OUTTopeniOkap2
#13 VzdalenyVystup11 <= OUTZasuvky1
#14 VzdalenyVystup12 <= OUTZasuvky3
#15 VzdalenyVystup13 <= OUTNouzoveOsvetleni
#16 VzdalenyVystup14 <= OUTVnitrniZasuvkyDenniProvoz
#17 VzdalenyVystup15 <= OUTVenkovniReklama
#18 VzdalenyVystup16 <= OUTTopeniOkap
#19 d2:D_klop(xVstup: VzdalenyVstup2)
#20 INVnitrniSvetla3 <= #21.xVystup
#21 d3:D_klop(xVstup: VzdalenyVstup3)
#22 INSvetloNadVchodem <= #23.xVystup
#23 d4:D_klop(xVstup: VzdalenyVstup4)
#24 INVnitrniZasuvkyDenniProvoz <= #25.xVystup
#25 d5:D_klop(xVstup: VzdalenyVstup5)
#26 INVnitrniReklama <= #27.xVystup
#27 d6:D_klop(xVstup: VzdalenyVstup6)
#28 INVenkovniReklama <= #29.xVystup
#29 d7:D_klop(xVstup: VzdalenyVstup7)
#30 INTopeniOkap <= #31.xVystup
#31 d8:D_klop(xVstup: VzdalenyVstup8)
#32 DIV(#34, 10.0)
#33 INVenkovniTeplota <= #32
#34 WORD_TO_REAL(VzdalenaTeplota1)
_END_CFC_
(* the same logic as Structured Text *)
VzdalenyVystup1 := OUTVnitrniSvetla1;
VzdalenyVystup2 := OUTVnitrniSvetla2;
VzdalenyVystup4 := OUTVnitrniReklama;
VzdalenyVystup5 := OUTVenkovniReklama1;
VzdalenyVystup6 := OUTVenkovniReklama2;
VzdalenyVystup7 := OUTVenkovniReklama3;
INVnitrniSvetla1 := d1.xVystup;
INVnitrniSvetla2 := d2.xVystup;
d1(xVstup := VzdalenyVstup1);
VzdalenyVystup3 := OUTVnitrniSvetla3;
VzdalenyVystup8 := OUTSvetloNadVchodem;
VzdalenyVystup9 := OUTTopeniOkap1;
VzdalenyVystup10 := OUTTopeniOkap2;
VzdalenyVystup11 := OUTZasuvky1;
VzdalenyVystup12 := OUTZasuvky3;
VzdalenyVystup13 := OUTNouzoveOsvetleni;
VzdalenyVystup14 := OUTVnitrniZasuvkyDenniProvoz;
VzdalenyVystup15 := OUTVenkovniReklama;
VzdalenyVystup16 := OUTTopeniOkap;
d2(xVstup := VzdalenyVstup2);
INVnitrniSvetla3 := d3.xVystup;
d3(xVstup := VzdalenyVstup3);
INSvetloNadVchodem := d4.xVystup;
d4(xVstup := VzdalenyVstup4);
INVnitrniZasuvkyDenniProvoz := d5.xVystup;
d5(xVstup := VzdalenyVstup5);
INVnitrniReklama := d6.xVystup;
d6(xVstup := VzdalenyVstup6);
INVenkovniReklama := d7.xVystup;
d7(xVstup := VzdalenyVstup7);
INTopeniOkap := d8.xVystup;
d8(xVstup := VzdalenyVstup8);
INVenkovniTeplota := _t91 / 10.0;
_t91 := WORD_TO_REAL(VzdalenaTeplota1);
END_PROGRAM

(* POU Ostatni/D_klop, ST *)
FUNCTION_BLOCK D_klop
VAR_INPUT
	xVstup: BOOL;
END_VAR
VAR_OUTPUT
	xVystup: BOOL;
END_VAR
VAR
	p: BOOL:= FALSE;
	a: BOOL:= TRUE;
END_VAR
IF(xVstup)
THEN
	IF(p)
	THEN
		IF (a)
			THEN
			xVystup := FALSE;
			p := FALSE;
			a := FALSE;
		END_IF
	ELSE
		IF (a)
			THEN
			xVystup := TRUE;
			p := TRUE;
			a := FALSE;
		END_IF
	END_IF
ELSE
	a:= TRUE;
END_IF
END_FUNCTION_BLOCK

(* POU ProdejnaMaterialu, FBD *)
PROGRAM ProdejnaMaterialu
VAR
	NEVIM: BOOL;
	zasuvky: IntervalSepnuti;
	PRGVnitrniZasuvkyDenniProvoz: BOOL;
	iZasuvkyStartHodiny: INT := 17;
	iZasuvkyStartMinuty: INT := 0;
	iZasuvkyKonecHodiny: INT := 6;
	iZasuvkyKonecMinuty: INT := 0;

	SvetloNadVchodem1: IntervalSepnuti;
	PRGSvetloNadVchodem: BOOL;
	iSvetloNadVchodemStartHodiny1: INT:= 8;
	iSvetloNadVchodemStartMinuty1: INT:= 0;
	iSvetloNadVchodemKonecHodiny1: INT:= 17;
	iSvetloNadVchodemKonecMinuty1: INT:= 0;
	rUrovenSvetlonadVchodem1: REAL;
	SvetloNadVchodem2: IntervalSepnuti;
	iSvetloNadVchodemStartHodiny2: INT:= 8;
	iSvetloNadVchodemStartMinuty2: INT:= 0;
	iSvetloNadVchodemKonecHodiny2: INT:= 17;
	iSvetloNadVchodemKonecMinuty2: INT:= 0;
	rUrovenSvetlonadVchodem2: REAL;
	xSvetloNadVchodemPracTyden: BOOL;
	xSvetloNadVchodemVikend: BOOL;

	iVnitrniReklamaStartHodiny1: INT:= 17;
	iVnitrniReklamaStartMinuty1: INT:= 0;
	iVnitrniReklamaKonecHodiny1: INT:= 22;
	iVnitrniReklamakonecMinuty1: INT:= 0;
	iVnitrniReklamaStartHodiny2: INT:= 5;
	iVnitrniReklamaStartMinuty2: INT:= 30;
	iVnitrniReklamaKonecHodiny2: INT:= 8;
	iVnitrniReklamakonecMinuty2: INT:= 0;
	NocniRezimVnitrniReklama1: IntervalSepnuti;
	NocniRezimVnitrniReklama2: IntervalSepnuti;
	PRGVnitrniReklama: BOOL;

	TeplotaVenkovniMAX: REAL:= 5.0;
	TeplotaVenkovniMIN: REAL:= -5.0;

	VnitrniSvetla1: IntervalSepnuti;
	VnitrniSvetla2: IntervalSepnuti;
	PRGVnitrniSvetla1: BOOL;
	iVnitrniSvetlaStartHodiny1: INT:= 6;
	iVnitrniSvetlaStartMinuty1: INT:= 45;
	iVnitrniSvetlaKonecHodiny1: INT:= 18;
	iVnitrniSvetlaKonecMinuty1: INT:= 0;
	rIntenzitaVnitrniSvetla1 : INT;
	iVnitrniSvetlaStartHodiny2: INT:= 6;
	iVnitrniSvetlaStartMinuty2: INT:= 45;
	iVnitrniSvetlaKonecHodiny2: INT:= 18;
	iVnitrniSvetlaKonecMinuty2: INT:= 0;
	rIntenzitaVnitrniSvetla2 : INT;
	xVnitrniSvetla1PracDen: BOOL;
	xVnitrniSvetla1Vikend: BOOL;

	VnitrniSvetla3: IntervalSepnuti;
	VnitrniSvetla4: IntervalSepnuti;
	PRGVnitrniSvetla2: BOOL;
	iVnitrniSvetlaStartHodiny3: INT:= 6;
	iVnitrniSvetlaStartMinuty3: INT:= 45;
	iVnitrniSvetlaKonecHodiny3: INT:= 18;
	iVnitrniSvetlaKonecMinuty3: INT:= 0;
	rIntenzitaVnitrniSvetla3 : INT;
	iVnitrniSvetlaStartHodiny4: INT:= 6;
	iVnitrniSvetlaStartMinuty4: INT:= 45;
	iVnitrniSvetlaKonecHodiny4: INT:= 18;
	iVnitrniSvetlaKonecMinuty4: INT:= 0;
	rIntenzitaVnitrniSvetla4 : INT;
	xVnitrniSvetla2PracDen: BOOL;
	xVnitrniSvetla2Vikend: BOOL;

	VnitrniSvetla5: IntervalSepnuti;
	VnitrniSvetla6: IntervalSepnuti;
	PRGVnitrniSvetla3: BOOL;
	iVnitrniSvetlaStartHodiny5: INT:= 6;
	iVnitrniSvetlaStartMinuty5: INT:= 45;
	iVnitrniSvetlaKonecHodiny5: INT:= 18;
	iVnitrniSvetlaKonecMinuty5: INT:= 0;
	rIntenzitaVnitrniSvetla5 : INT;
	iVnitrniSvetlaStartHodiny6: INT:= 6;
	iVnitrniSvetlaStartMinuty6: INT:= 45;
	iVnitrniSvetlaKonecHodiny6: INT:= 18;
	iVnitrniSvetlaKonecMinuty6: INT:= 0;
	rIntenzitaVnitrniSvetla6 : INT;
	xVnitrniSvetla3PracDen: BOOL;
	xVnitrniSvetla3Vikend: BOOL;
END_VAR
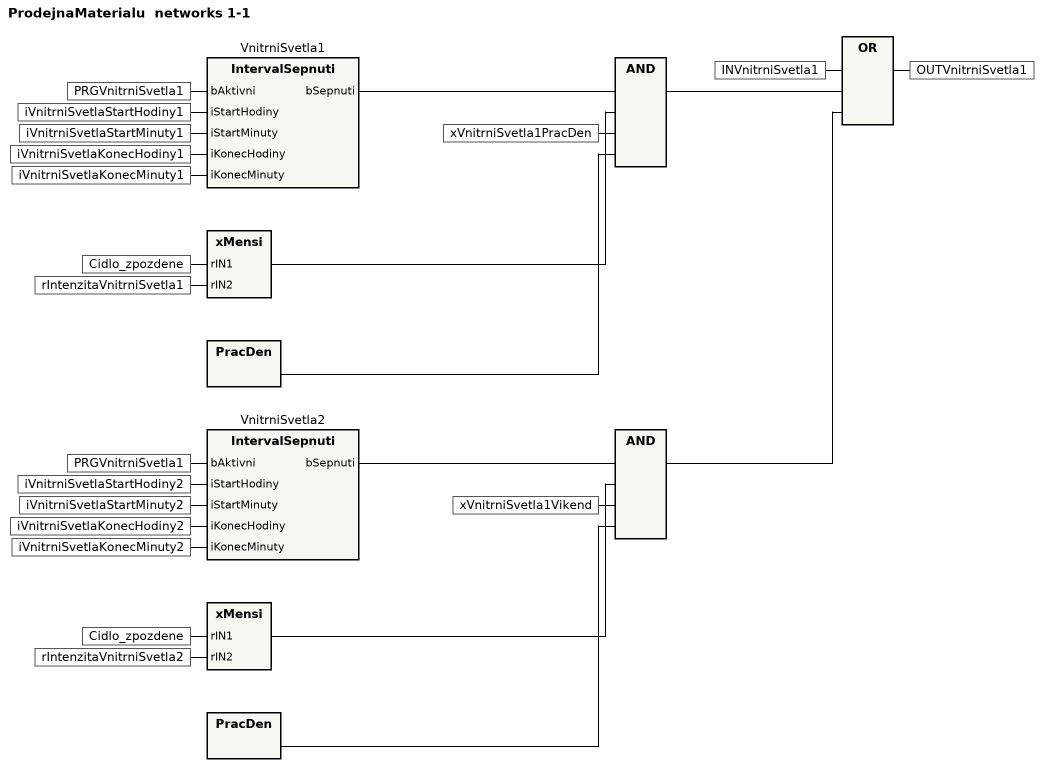
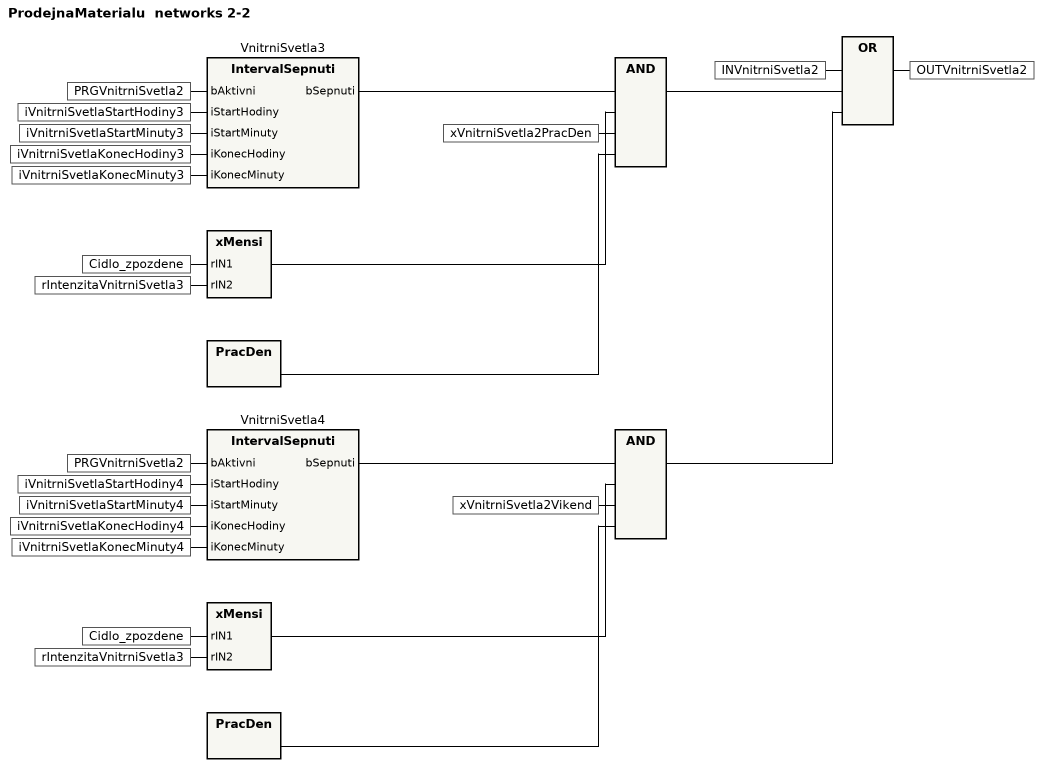
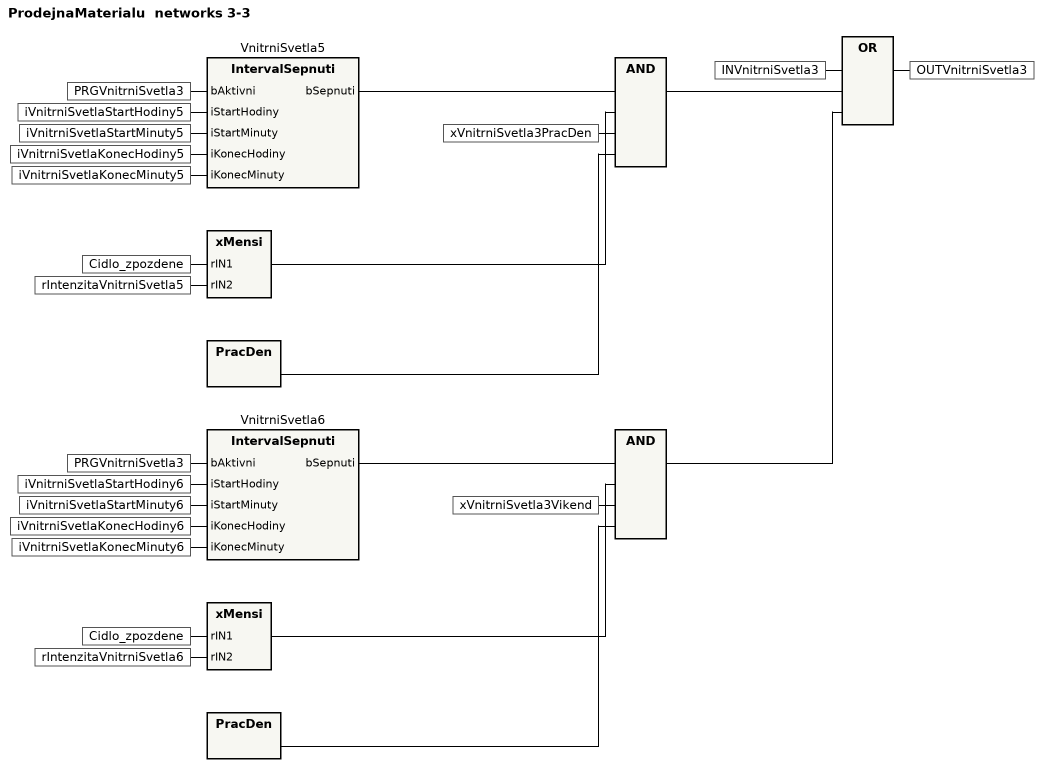
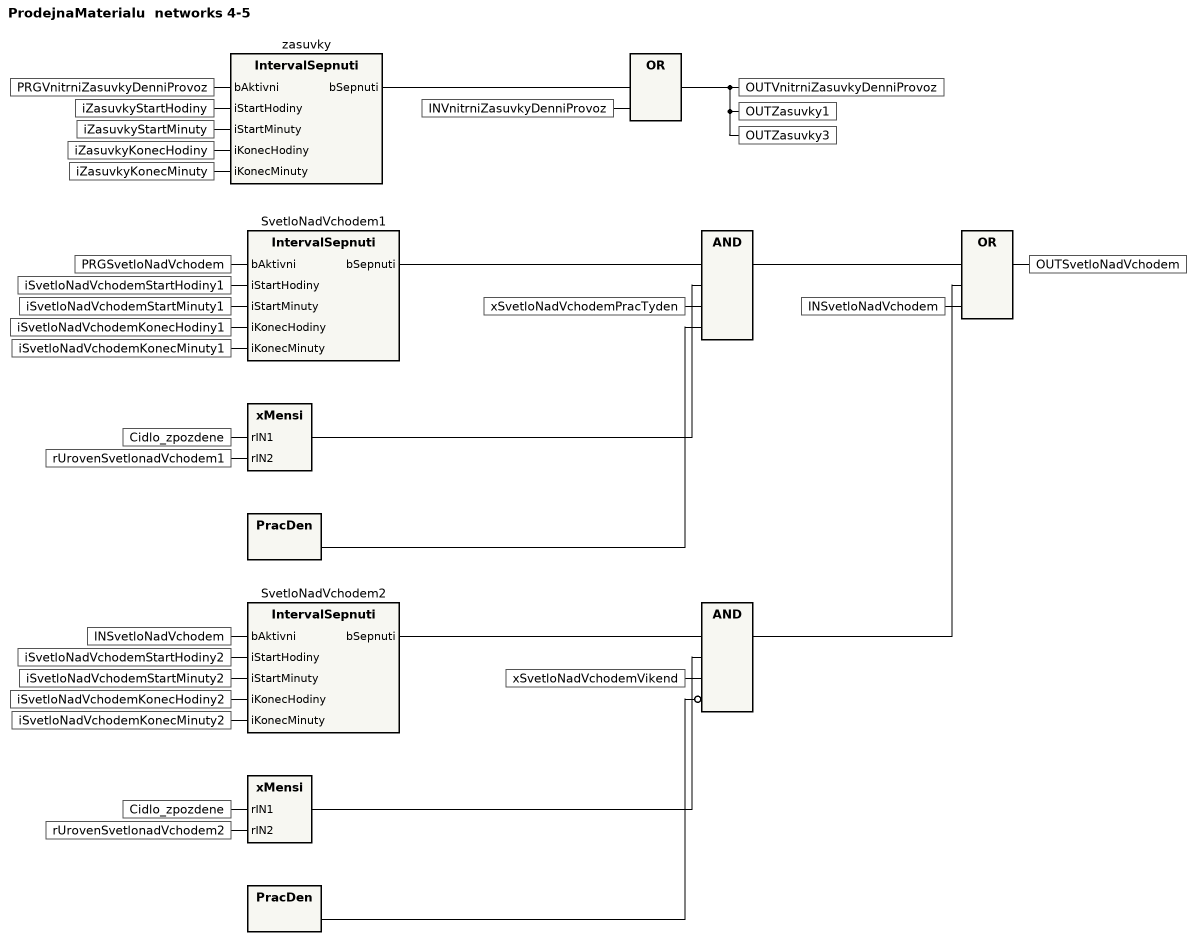
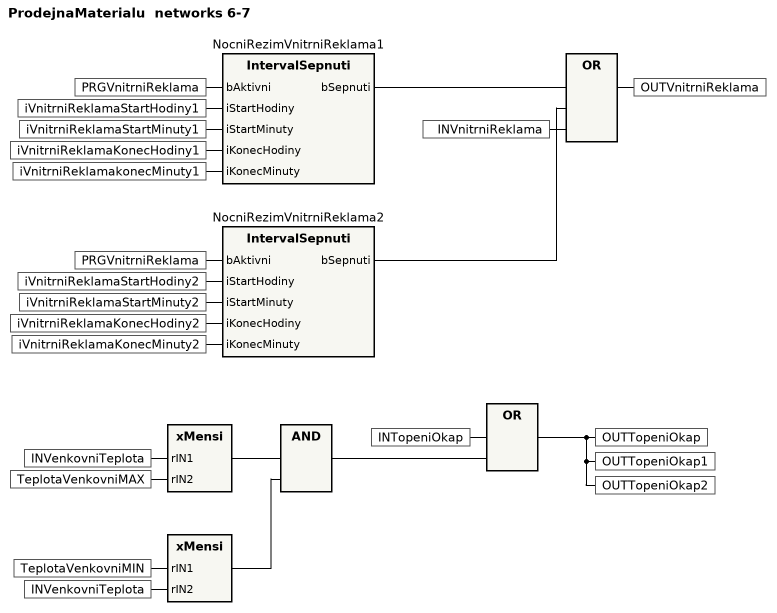
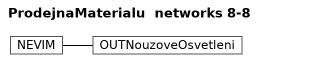
_FBD_ (* Function Block Diagram *)
NETWORK 1
	OR(INVnitrniSvetla1, AND(VnitrniSvetla1:IntervalSepnuti(bAktivni: PRGVnitrniSvetla1, iStartHodiny: iVnitrniSvetlaStartHodiny1, iStartMinuty: iVnitrniSvetlaStartMinuty1, iKonecHodiny: iVnitrniSvetlaKonecHodiny1, iKonecMinuty: iVnitrniSvetlaKonecMinuty1), xMensi(rIN1: Cidlo_zpozdene, rIN2: rIntenzitaVnitrniSvetla1), xVnitrniSvetla1PracDen, PracDen()), AND(VnitrniSvetla2:IntervalSepnuti(bAktivni: PRGVnitrniSvetla1, iStartHodiny: iVnitrniSvetlaStartHodiny2, iStartMinuty: iVnitrniSvetlaStartMinuty2, iKonecHodiny: iVnitrniSvetlaKonecHodiny2, iKonecMinuty: iVnitrniSvetlaKonecMinuty2), xMensi(rIN1: Cidlo_zpozdene, rIN2: rIntenzitaVnitrniSvetla2), xVnitrniSvetla1Vikend, PracDen())) => OUTVnitrniSvetla1
NETWORK 2
	OR(INVnitrniSvetla2, AND(VnitrniSvetla3:IntervalSepnuti(bAktivni: PRGVnitrniSvetla2, iStartHodiny: iVnitrniSvetlaStartHodiny3, iStartMinuty: iVnitrniSvetlaStartMinuty3, iKonecHodiny: iVnitrniSvetlaKonecHodiny3, iKonecMinuty: iVnitrniSvetlaKonecMinuty3), xMensi(rIN1: Cidlo_zpozdene, rIN2: rIntenzitaVnitrniSvetla3), xVnitrniSvetla2PracDen, PracDen()), AND(VnitrniSvetla4:IntervalSepnuti(bAktivni: PRGVnitrniSvetla2, iStartHodiny: iVnitrniSvetlaStartHodiny4, iStartMinuty: iVnitrniSvetlaStartMinuty4, iKonecHodiny: iVnitrniSvetlaKonecHodiny4, iKonecMinuty: iVnitrniSvetlaKonecMinuty4), xMensi(rIN1: Cidlo_zpozdene, rIN2: rIntenzitaVnitrniSvetla3), xVnitrniSvetla2Vikend, PracDen())) => OUTVnitrniSvetla2
NETWORK 3
	OR(INVnitrniSvetla3, AND(VnitrniSvetla5:IntervalSepnuti(bAktivni: PRGVnitrniSvetla3, iStartHodiny: iVnitrniSvetlaStartHodiny5, iStartMinuty: iVnitrniSvetlaStartMinuty5, iKonecHodiny: iVnitrniSvetlaKonecHodiny5, iKonecMinuty: iVnitrniSvetlaKonecMinuty5), xMensi(rIN1: Cidlo_zpozdene, rIN2: rIntenzitaVnitrniSvetla5), xVnitrniSvetla3PracDen, PracDen()), AND(VnitrniSvetla6:IntervalSepnuti(bAktivni: PRGVnitrniSvetla3, iStartHodiny: iVnitrniSvetlaStartHodiny6, iStartMinuty: iVnitrniSvetlaStartMinuty6, iKonecHodiny: iVnitrniSvetlaKonecHodiny6, iKonecMinuty: iVnitrniSvetlaKonecMinuty6), xMensi(rIN1: Cidlo_zpozdene, rIN2: rIntenzitaVnitrniSvetla6), xVnitrniSvetla3Vikend, PracDen())) => OUTVnitrniSvetla3
NETWORK 4
	OR(zasuvky:IntervalSepnuti(bAktivni: PRGVnitrniZasuvkyDenniProvoz, iStartHodiny: iZasuvkyStartHodiny, iStartMinuty: iZasuvkyStartMinuty, iKonecHodiny: iZasuvkyKonecHodiny, iKonecMinuty: iZasuvkyKonecMinuty), INVnitrniZasuvkyDenniProvoz) => OUTVnitrniZasuvkyDenniProvoz, OUTZasuvky1, OUTZasuvky3
NETWORK 5
	OR(AND(SvetloNadVchodem1:IntervalSepnuti(bAktivni: PRGSvetloNadVchodem, iStartHodiny: iSvetloNadVchodemStartHodiny1, iStartMinuty: iSvetloNadVchodemStartMinuty1, iKonecHodiny: iSvetloNadVchodemKonecHodiny1, iKonecMinuty: iSvetloNadVchodemKonecMinuty1), xMensi(rIN1: Cidlo_zpozdene, rIN2: rUrovenSvetlonadVchodem1), xSvetloNadVchodemPracTyden, PracDen()), AND(SvetloNadVchodem2:IntervalSepnuti(bAktivni: INSvetloNadVchodem, iStartHodiny: iSvetloNadVchodemStartHodiny2, iStartMinuty: iSvetloNadVchodemStartMinuty2, iKonecHodiny: iSvetloNadVchodemKonecHodiny2, iKonecMinuty: iSvetloNadVchodemKonecMinuty2), xMensi(rIN1: Cidlo_zpozdene, rIN2: rUrovenSvetlonadVchodem2), xSvetloNadVchodemVikend, NOT PracDen()), INSvetloNadVchodem) => OUTSvetloNadVchodem
NETWORK 6
	OR(NocniRezimVnitrniReklama1:IntervalSepnuti(bAktivni: PRGVnitrniReklama, iStartHodiny: iVnitrniReklamaStartHodiny1, iStartMinuty: iVnitrniReklamaStartMinuty1, iKonecHodiny: iVnitrniReklamaKonecHodiny1, iKonecMinuty: iVnitrniReklamakonecMinuty1), NocniRezimVnitrniReklama2:IntervalSepnuti(bAktivni: PRGVnitrniReklama, iStartHodiny: iVnitrniReklamaStartHodiny2, iStartMinuty: iVnitrniReklamaStartMinuty2, iKonecHodiny: iVnitrniReklamaKonecHodiny2, iKonecMinuty: iVnitrniReklamaKonecMinuty2), 	INVnitrniReklama) => OUTVnitrniReklama
NETWORK 7
	OR(INTopeniOkap, AND(xMensi(rIN1: INVenkovniTeplota, rIN2: TeplotaVenkovniMAX), xMensi(rIN1: TeplotaVenkovniMIN, rIN2: INVenkovniTeplota))) => OUTTopeniOkap, OUTTopeniOkap1, OUTTopeniOkap2
NETWORK 8
	NEVIM => OUTNouzoveOsvetleni
_END_FBD_
(* the same logic as Structured Text *)
(* Network 1 *)
VnitrniSvetla1(bAktivni := PRGVnitrniSvetla1, iStartHodiny := iVnitrniSvetlaStartHodiny1, iStartMinuty := iVnitrniSvetlaStartMinuty1, iKonecHodiny := iVnitrniSvetlaKonecHodiny1, iKonecMinuty := iVnitrniSvetlaKonecMinuty1);
VnitrniSvetla2(bAktivni := PRGVnitrniSvetla1, iStartHodiny := iVnitrniSvetlaStartHodiny2, iStartMinuty := iVnitrniSvetlaStartMinuty2, iKonecHodiny := iVnitrniSvetlaKonecHodiny2, iKonecMinuty := iVnitrniSvetlaKonecMinuty2);
OUTVnitrniSvetla1 := INVnitrniSvetla1 OR (VnitrniSvetla1.bSepnuti AND xMensi(rIN1 := Cidlo_zpozdene, rIN2 := rIntenzitaVnitrniSvetla1) AND xVnitrniSvetla1PracDen AND PracDen()) OR (VnitrniSvetla2.bSepnuti AND xMensi(rIN1 := Cidlo_zpozdene, rIN2 := rIntenzitaVnitrniSvetla2) AND xVnitrniSvetla1Vikend AND PracDen());
(* Network 2 *)
VnitrniSvetla3(bAktivni := PRGVnitrniSvetla2, iStartHodiny := iVnitrniSvetlaStartHodiny3, iStartMinuty := iVnitrniSvetlaStartMinuty3, iKonecHodiny := iVnitrniSvetlaKonecHodiny3, iKonecMinuty := iVnitrniSvetlaKonecMinuty3);
VnitrniSvetla4(bAktivni := PRGVnitrniSvetla2, iStartHodiny := iVnitrniSvetlaStartHodiny4, iStartMinuty := iVnitrniSvetlaStartMinuty4, iKonecHodiny := iVnitrniSvetlaKonecHodiny4, iKonecMinuty := iVnitrniSvetlaKonecMinuty4);
OUTVnitrniSvetla2 := INVnitrniSvetla2 OR (VnitrniSvetla3.bSepnuti AND xMensi(rIN1 := Cidlo_zpozdene, rIN2 := rIntenzitaVnitrniSvetla3) AND xVnitrniSvetla2PracDen AND PracDen()) OR (VnitrniSvetla4.bSepnuti AND xMensi(rIN1 := Cidlo_zpozdene, rIN2 := rIntenzitaVnitrniSvetla3) AND xVnitrniSvetla2Vikend AND PracDen());
(* Network 3 *)
VnitrniSvetla5(bAktivni := PRGVnitrniSvetla3, iStartHodiny := iVnitrniSvetlaStartHodiny5, iStartMinuty := iVnitrniSvetlaStartMinuty5, iKonecHodiny := iVnitrniSvetlaKonecHodiny5, iKonecMinuty := iVnitrniSvetlaKonecMinuty5);
VnitrniSvetla6(bAktivni := PRGVnitrniSvetla3, iStartHodiny := iVnitrniSvetlaStartHodiny6, iStartMinuty := iVnitrniSvetlaStartMinuty6, iKonecHodiny := iVnitrniSvetlaKonecHodiny6, iKonecMinuty := iVnitrniSvetlaKonecMinuty6);
OUTVnitrniSvetla3 := INVnitrniSvetla3 OR (VnitrniSvetla5.bSepnuti AND xMensi(rIN1 := Cidlo_zpozdene, rIN2 := rIntenzitaVnitrniSvetla5) AND xVnitrniSvetla3PracDen AND PracDen()) OR (VnitrniSvetla6.bSepnuti AND xMensi(rIN1 := Cidlo_zpozdene, rIN2 := rIntenzitaVnitrniSvetla6) AND xVnitrniSvetla3Vikend AND PracDen());
(* Network 4 *)
zasuvky(bAktivni := PRGVnitrniZasuvkyDenniProvoz, iStartHodiny := iZasuvkyStartHodiny, iStartMinuty := iZasuvkyStartMinuty, iKonecHodiny := iZasuvkyKonecHodiny, iKonecMinuty := iZasuvkyKonecMinuty);
OUTVnitrniZasuvkyDenniProvoz := zasuvky.bSepnuti OR INVnitrniZasuvkyDenniProvoz;
OUTZasuvky1 := OUTVnitrniZasuvkyDenniProvoz;
OUTZasuvky3 := OUTVnitrniZasuvkyDenniProvoz;
(* Network 5 *)
SvetloNadVchodem1(bAktivni := PRGSvetloNadVchodem, iStartHodiny := iSvetloNadVchodemStartHodiny1, iStartMinuty := iSvetloNadVchodemStartMinuty1, iKonecHodiny := iSvetloNadVchodemKonecHodiny1, iKonecMinuty := iSvetloNadVchodemKonecMinuty1);
SvetloNadVchodem2(bAktivni := INSvetloNadVchodem, iStartHodiny := iSvetloNadVchodemStartHodiny2, iStartMinuty := iSvetloNadVchodemStartMinuty2, iKonecHodiny := iSvetloNadVchodemKonecHodiny2, iKonecMinuty := iSvetloNadVchodemKonecMinuty2);
OUTSvetloNadVchodem := (SvetloNadVchodem1.bSepnuti AND xMensi(rIN1 := Cidlo_zpozdene, rIN2 := rUrovenSvetlonadVchodem1) AND xSvetloNadVchodemPracTyden AND PracDen()) OR (SvetloNadVchodem2.bSepnuti AND xMensi(rIN1 := Cidlo_zpozdene, rIN2 := rUrovenSvetlonadVchodem2) AND xSvetloNadVchodemVikend AND NOT PracDen()) OR INSvetloNadVchodem;
(* Network 6 *)
NocniRezimVnitrniReklama1(bAktivni := PRGVnitrniReklama, iStartHodiny := iVnitrniReklamaStartHodiny1, iStartMinuty := iVnitrniReklamaStartMinuty1, iKonecHodiny := iVnitrniReklamaKonecHodiny1, iKonecMinuty := iVnitrniReklamakonecMinuty1);
NocniRezimVnitrniReklama2(bAktivni := PRGVnitrniReklama, iStartHodiny := iVnitrniReklamaStartHodiny2, iStartMinuty := iVnitrniReklamaStartMinuty2, iKonecHodiny := iVnitrniReklamaKonecHodiny2, iKonecMinuty := iVnitrniReklamaKonecMinuty2);
OUTVnitrniReklama := NocniRezimVnitrniReklama1.bSepnuti OR NocniRezimVnitrniReklama2.bSepnuti OR (	INVnitrniReklama);
(* Network 7 *)
OUTTopeniOkap := INTopeniOkap OR (xMensi(rIN1 := INVenkovniTeplota, rIN2 := TeplotaVenkovniMAX) AND xMensi(rIN1 := TeplotaVenkovniMIN, rIN2 := INVenkovniTeplota));
OUTTopeniOkap1 := OUTTopeniOkap;
OUTTopeniOkap2 := OUTTopeniOkap;
(* Network 8 *)
OUTNouzoveOsvetleni := NEVIM;
END_PROGRAM

(* POU Ostatni/IntervalSepnuti, ST *)
FUNCTION_BLOCK IntervalSepnuti
VAR_INPUT
	bAktivni: BOOL;
	iStartHodiny: INT;
	iStartMinuty: INT;
	iKonecHodiny: INT;
	iKonecMinuty: INT;
END_VAR
VAR_OUTPUT
	bSepnuti: BOOL;
END_VAR
VAR
END_VAR
IF (bAktivni)
THEN
	IF(iStartHodiny = PLC_PRG.System_datum.Hour )
	THEN
		IF(iStartMinuty <= PLC_PRG.System_datum.Minute)
		THEN
			bSepnuti:= TRUE;
		END_IF
	ELSIF (iStartHodiny < PLC_PRG.System_datum.Hour)
	THEN
		bSepnuti := TRUE;
	ELSE
		bSepnuti := FALSE;
	END_IF

	IF(iKonecHodiny = PLC_PRG.System_datum.Hour)
	THEN
		IF(iKonecMinuty <= PLC_PRG.System_datum.Minute)
		THEN
			bSepnuti := FALSE;
		END_IF

	ELSIF(iKonecHodiny < PLC_PRG.System_datum.Hour)
	THEN
		bSepnuti := FALSE;
	ELSE
		bSepnuti := TRUE;
	END_IF
END_IF
END_FUNCTION_BLOCK

(* POU Ostatni/xMensi, ST *)
FUNCTION xMensi : BOOL
VAR_INPUT
	rIN1: REAL;
	rIN2: REAL;
END_VAR
VAR
END_VAR
IF(rIN1<rIN2)
THEN
	xMensi := TRUE;
ELSE
	xMensi := FALSE;
END_IF
END_FUNCTION

(* POU Ostatni/PracDen, ST *)
FUNCTION PracDen : BOOL
VAR_INPUT
END_VAR
VAR
	datum: SystemTimeDate;
END_VAR
IF ((datum.DayOfWeek = 6) OR (datum.DayOfWeek = 7))
THEN
	PracDen := FALSE;
ELSE
	PracDen := TRUE;
END_IF
END_FUNCTION

(* POU Ostatni/LetniZimniCas, FBD *)
PROGRAM LetniZimniCas
VAR
	sCasDatumPomoc: STRING;
END_VAR
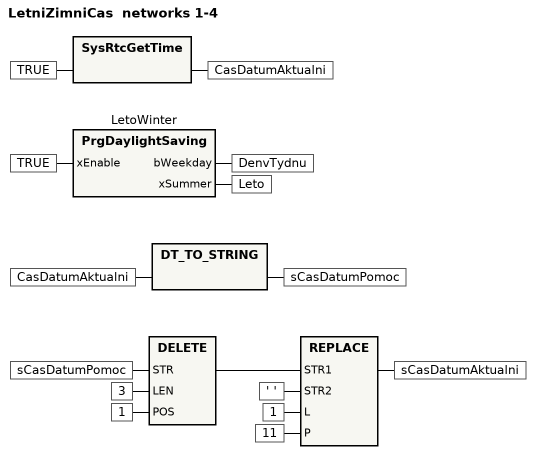
_FBD_ (* Function Block Diagram *)
NETWORK 1 (* Prwcti aktualni datum v procesoru *)
	SysRtcGetTime(TRUE) => CasDatumAktualni
NETWORK 2 (* Automaticky prechod z letniho na zimni cas / DenvTydnu: Pondeli = 1; Utery = 2; Streda = 3; Ctvrtek = 4; Patek = 5; Sobota = 6; Nedele = 7 *)
	LetoWinter:PrgDaylightSaving(xEnable: TRUE, xSummer => Leto) => DenvTydnu
NETWORK 3
	DT_TO_STRING(CasDatumAktualni) => sCasDatumPomoc
NETWORK 4
	REPLACE(STR1: DELETE(STR: sCasDatumPomoc, LEN: 3, POS: 1), STR2: ' ', L: 1, P: 11) => sCasDatumAktualni
_END_FBD_
(* the same logic as Structured Text *)
(* Network 1: Prwcti aktualni datum v procesoru *)
CasDatumAktualni := SysRtcGetTime(TRUE);
(* Network 2: Automaticky prechod z letniho na zimni cas / DenvTydnu: Pondeli = 1; Utery = 2; Streda = 3; Ctvrtek = 4; Patek = 5; Sobota = 6; Nedele = 7 *)
LetoWinter(xEnable := TRUE);
Leto := LetoWinter.xSummer;
DenvTydnu := LetoWinter.bWeekday;
(* Network 3 *)
sCasDatumPomoc := DT_TO_STRING(CasDatumAktualni);
(* Network 4 *)
sCasDatumAktualni := REPLACE(DELETE(sCasDatumPomoc, 3, 1), ' ', 1, 11);
END_PROGRAM

(* POU Ostatni/CasProg, CFC *)
PROGRAM CasProg
VAR
	CasProg1: FbScheduleWeekly;
	CasProg2: FbScheduleWeekly;

	CasProg3: FbScheduleWeekly;
	CasProg4: FbScheduleWeekly;

	CasProg5: FbScheduleWeekly;
	CasProg6: FbScheduleWeekly;
END_VAR
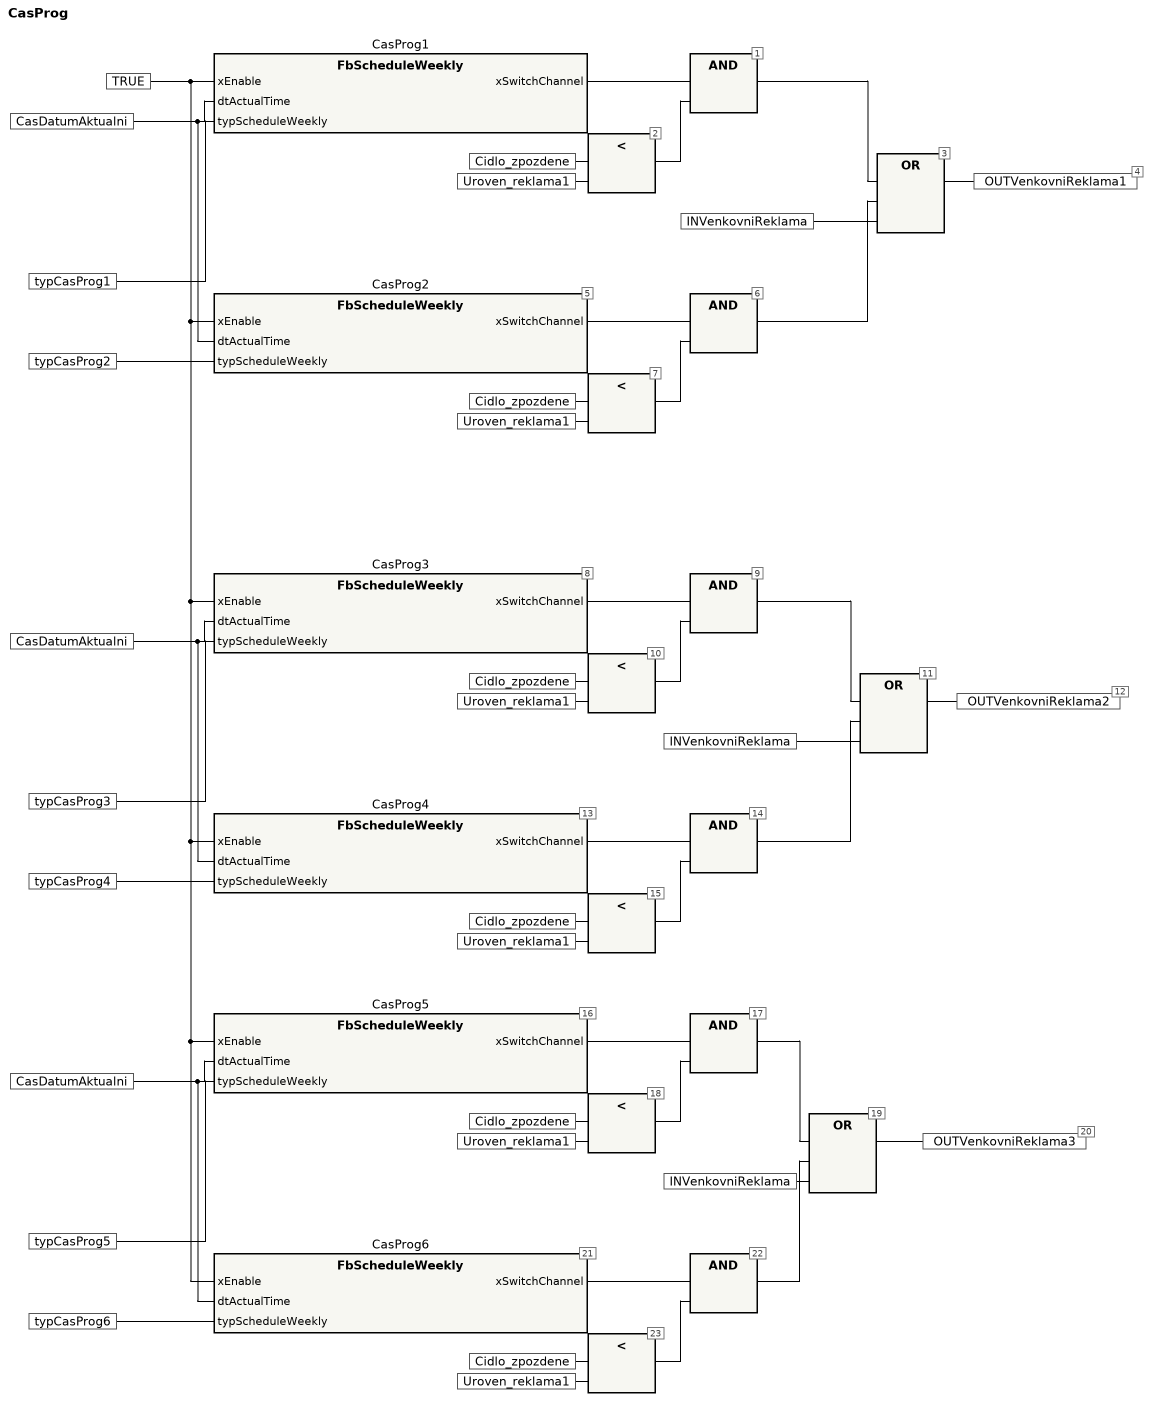
_CFC_ (* Continuous Function Chart, elements in execution order *)
#0 CasProg1:FbScheduleWeekly(xEnable: TRUE, dtActualTime: CasDatumAktualni, typScheduleWeekly: typCasProg1)
#1 AND(#0.xSwitchChannel, #2)
#2 <(Cidlo_zpozdene, Uroven_reklama1)
#3 OR(#1, #6, INVenkovniReklama)
#4 OUTVenkovniReklama1 <= #3
#5 CasProg2:FbScheduleWeekly(xEnable: TRUE, dtActualTime: CasDatumAktualni, typScheduleWeekly: typCasProg2)
#6 AND(#5.xSwitchChannel, #7)
#7 <(Cidlo_zpozdene, Uroven_reklama1)
#8 CasProg3:FbScheduleWeekly(xEnable: TRUE, dtActualTime: CasDatumAktualni, typScheduleWeekly: typCasProg3)
#9 AND(#8.xSwitchChannel, #10)
#10 <(Cidlo_zpozdene, Uroven_reklama1)
#11 OR(#9, #14, INVenkovniReklama)
#12 OUTVenkovniReklama2 <= #11
#13 CasProg4:FbScheduleWeekly(xEnable: TRUE, dtActualTime: CasDatumAktualni, typScheduleWeekly: typCasProg4)
#14 AND(#13.xSwitchChannel, #15)
#15 <(Cidlo_zpozdene, Uroven_reklama1)
#16 CasProg5:FbScheduleWeekly(xEnable: TRUE, dtActualTime: CasDatumAktualni, typScheduleWeekly: typCasProg5)
#17 AND(#16.xSwitchChannel, #18)
#18 <(Cidlo_zpozdene, Uroven_reklama1)
#19 OR(#17, #22, INVenkovniReklama)
#20 OUTVenkovniReklama3 <= #19
#21 CasProg6:FbScheduleWeekly(xEnable: TRUE, dtActualTime: CasDatumAktualni, typScheduleWeekly: typCasProg6)
#22 AND(#21.xSwitchChannel, #23)
#23 <(Cidlo_zpozdene, Uroven_reklama1)
_END_CFC_
END_PROGRAM

(* POU Kolotoc/DlouhyStisk, CFC *)
PROGRAM DlouhyStisk
VAR_INPUT
	Vstup: BOOL;
END_VAR
VAR_OUTPUT
	DlouhyS: BOOL;
	KratkyS: BOOL;
END_VAR
VAR
	cas1: TON;
	cas2: TOF;
	cas3: TON;
	cas4: TOF;
END_VAR
VAR (* helpers for the ST form of the networks *)
	_t57 : BOOL;
END_VAR
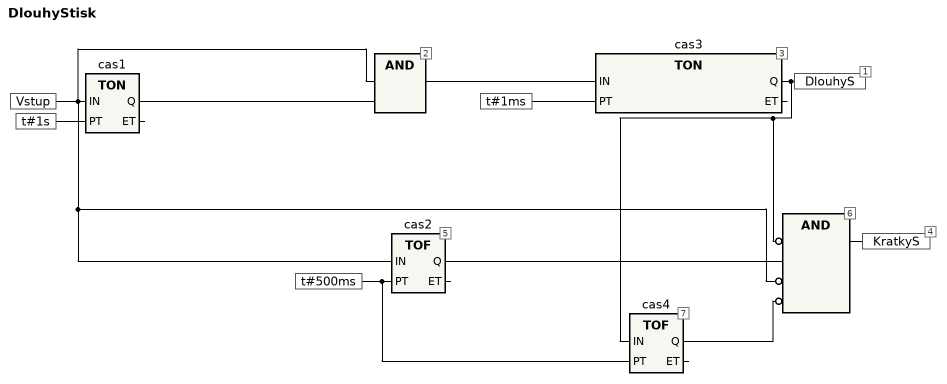
_CFC_ (* Continuous Function Chart, elements in execution order *)
#0 cas1:TON(IN: Vstup, PT: t#1s)
#1 DlouhyS <= #3.Q
#2 AND(Vstup, #0.Q)
#3 cas3:TON(IN: #2, PT: t#1ms)
#4 KratkyS <= #6
#5 cas2:TOF(IN: Vstup, PT: t#500ms)
#6 AND(NOT #3.Q, #5.Q, NOT Vstup, NOT #7.Q)
#7 cas4:TOF(IN: #3.Q, PT: t#500ms)
_END_CFC_
(* the same logic as Structured Text *)
cas1(IN := Vstup, PT := t#1s);
DlouhyS := cas3.Q;
cas3(IN := Vstup AND cas1.Q, PT := t#1ms);
KratkyS := _t57;
cas2(IN := Vstup, PT := t#500ms);
_t57 := NOT cas3.Q AND cas2.Q AND NOT Vstup AND NOT cas4.Q;
cas4(IN := cas3.Q, PT := t#500ms);
END_PROGRAM

(* POU Kolotoc/DlouhyStisk2, CFC *)
PROGRAM DlouhyStisk2
VAR_INPUT
	Vstup: BOOL;
END_VAR
VAR_OUTPUT
	DlouhyS: BOOL;
	KratkyS: BOOL;
END_VAR
VAR
	cas1: TON;
	cas2: TOF;
	cas3: TON;
	cas4: TOF;
END_VAR
VAR (* helpers for the ST form of the networks *)
	_t57 : BOOL;
END_VAR
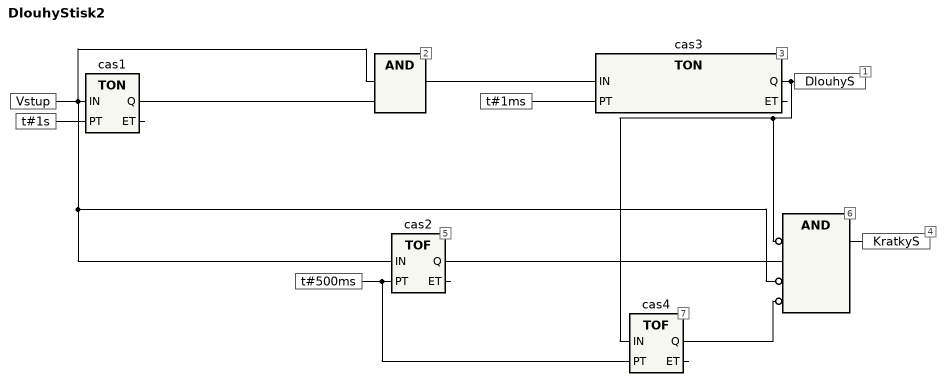
_CFC_ (* Continuous Function Chart, elements in execution order *)
#0 cas1:TON(IN: Vstup, PT: t#1s)
#1 DlouhyS <= #3.Q
#2 AND(Vstup, #0.Q)
#3 cas3:TON(IN: #2, PT: t#1ms)
#4 KratkyS <= #6
#5 cas2:TOF(IN: Vstup, PT: t#500ms)
#6 AND(NOT #3.Q, #5.Q, NOT Vstup, NOT #7.Q)
#7 cas4:TOF(IN: #3.Q, PT: t#500ms)
_END_CFC_
(* the same logic as Structured Text *)
cas1(IN := Vstup, PT := t#1s);
DlouhyS := cas3.Q;
cas3(IN := Vstup AND cas1.Q, PT := t#1ms);
KratkyS := _t57;
cas2(IN := Vstup, PT := t#500ms);
_t57 := NOT cas3.Q AND cas2.Q AND NOT Vstup AND NOT cas4.Q;
cas4(IN := cas3.Q, PT := t#500ms);
END_PROGRAM

(* POU Kolotoc/KolotocM, ST *)
PROGRAM KolotocM
VAR
	index: INT := 0;
	a: BOOL := FALSE;
	b: BOOL := FALSE;
END_VAR
VAR_INPUT
	KratkyStiskPlus: BOOL;
	KratkyStiskMinus: BOOL;
	DlouhyStiskPlus: BOOL;
	DlouhyStiskMinus: BOOL;
	PocetAktivnichVystupu: INT;
END_VAR
VAR_OUTPUT
	Rele1: BOOL;
	Rele2: BOOL;
	Rele3: BOOL;
	Rele4: BOOL;
	Rele5: BOOL;
	Rele6: BOOL;
	Rele7: BOOL;
	Rele8: BOOL;
	Rele9: BOOL;
	Rele10: BOOL;
	Rele11: BOOL;
	Rele12: BOOL;
END_VAR
IF (KratkyStiskPlus)
THEN
	a := TRUE;
END_IF

IF (a AND KratkyStiskPlus = FALSE)
	THEN
	index := index + 1;
	a := FALSE;
END_IF

IF (KratkyStiskMinus)
THEN
	b := TRUE;
END_IF

IF (b AND KratkyStiskMinus = FALSE)
THEN
	index := index - 1;
	b := FALSE;
END_IF

IF (index = -1)
THEN
	index := PocetAktivnichVystupu;
END_IF

IF (index = PocetAktivnichVystupu + 1)
THEN
	index := 0;
END_IF

IF (index = 0 )
THEN
	Rele1 := FALSE;
	Rele2 := FALSE;
	Rele3 := FALSE;
	Rele4 := FALSE;
	Rele5 := FALSE;
	Rele6 := FALSE;
	Rele7 := FALSE;
	Rele8 := FALSE;
	Rele9 := FALSE;
	Rele10 := FALSE;
	Rele11 := FALSE;
	Rele12 := FALSE;
ELSIF (index = 1)
THEN
	Rele1 := TRUE;
	Rele2 := FALSE;
	Rele3 := FALSE;
	Rele4 := FALSE;
	Rele5 := FALSE;
	Rele6 := FALSE;
	Rele7 := FALSE;
	Rele8 := FALSE;
	Rele9 := FALSE;
	Rele10 := FALSE;
ELSIF (index = 2)
THEN
	Rele1 := FALSE;
	Rele2 := TRUE;
	Rele3 := FALSE;
	Rele4 := FALSE;
	Rele5 := FALSE;
	Rele6 := FALSE;
	Rele7 := FALSE;
	Rele8 := FALSE;
	Rele9 := FALSE;
	Rele10 := FALSE;
	Rele11 := FALSE;
	Rele12 := FALSE;
ELSIF (index = 3)
THEN
	Rele1 := FALSE;
	Rele2 := FALSE;
	Rele3 := TRUE;
	Rele4 := FALSE;
	Rele5 := FALSE;
	Rele6 := FALSE;
	Rele7 := FALSE;
	Rele8 := FALSE;
	Rele9 := FALSE;
	Rele10 := FALSE;
	Rele11 := FALSE;
	Rele12 := FALSE;
ELSIF (index = 4)
THEN
	Rele1 := FALSE;
	Rele2 := FALSE;
	Rele3 := FALSE;
	Rele4 := TRUE;
	Rele5 := FALSE;
	Rele6 := FALSE;
	Rele7 := FALSE;
	Rele8 := FALSE;
	Rele9 := FALSE;
	Rele10 := FALSE;
	Rele11 := FALSE;
	Rele12 := FALSE;
ELSIF (index = 5)
THEN
	Rele1 := FALSE;
	Rele2 := FALSE;
	Rele3 := FALSE;
	Rele4 := FALSE;
	Rele5 := TRUE;
	Rele6 := FALSE;
	Rele7 := FALSE;
	Rele8 := FALSE;
	Rele9 := FALSE;
	Rele10 := FALSE;
	Rele11 := FALSE;
	Rele12 := FALSE;
ELSIF (index = 6)
THEN
	Rele1 := FALSE;
	Rele2 := FALSE;
	Rele3 := FALSE;
	Rele4 := FALSE;
	Rele5 := FALSE;
	Rele6 := TRUE;
	Rele7 := FALSE;
	Rele8 := FALSE;
	Rele9 := FALSE;
	Rele10 := FALSE;
	Rele11 := FALSE;
	Rele12 := FALSE;
ELSIF (index = 7)
THEN
	Rele1 := FALSE;
	Rele2 := FALSE;
	Rele3 := FALSE;
	Rele4 := FALSE;
	Rele5 := FALSE;
	Rele6 := FALSE;
	Rele7 := TRUE;
	Rele8 := FALSE;
	Rele9 := FALSE;
	Rele10 := FALSE;
	Rele11 := FALSE;
	Rele12 := FALSE;
ELSIF (index = 8)
THEN
	Rele1 := FALSE;
	Rele2 := FALSE;
	Rele3 := FALSE;
	Rele4 := FALSE;
	Rele5 := FALSE;
	Rele6 := FALSE;
	Rele7 := FALSE;
	Rele8 := TRUE;
	Rele9 := FALSE;
	Rele10 := FALSE;
	Rele11 := FALSE;
	Rele12 := FALSE;
ELSIF (index = 9)
THEN
	Rele1 := FALSE;
	Rele2 := FALSE;
	Rele3 := FALSE;
	Rele4 := FALSE;
	Rele5 := FALSE;
	Rele6 := FALSE;
	Rele7 := FALSE;
	Rele8 := FALSE;
	Rele9 := TRUE;
	Rele10 := FALSE;
	Rele11 := FALSE;
	Rele12 := FALSE;
ELSIF (index = 10)
THEN
	Rele1 := FALSE;
	Rele2 := FALSE;
	Rele3 := FALSE;
	Rele4 := FALSE;
	Rele5 := FALSE;
	Rele6 := FALSE;
	Rele7 := FALSE;
	Rele8 := FALSE;
	Rele9 := FALSE;
	Rele10 := TRUE;
	Rele11 := FALSE;
	Rele12 := FALSE;
ELSIF (index = 11)
THEN
	Rele1 := FALSE;
	Rele2 := FALSE;
	Rele3 := FALSE;
	Rele4 := FALSE;
	Rele5 := FALSE;
	Rele6 := FALSE;
	Rele7 := FALSE;
	Rele8 := FALSE;
	Rele9 := FALSE;
	Rele10 := FALSE;
	Rele11 := TRUE;
	Rele12 := FALSE;
ELSIF (index = 12)
THEN
	Rele1 := FALSE;
	Rele2 := FALSE;
	Rele3 := FALSE;
	Rele4 := FALSE;
	Rele5 := FALSE;
	Rele6 := FALSE;
	Rele7 := FALSE;
	Rele8 := FALSE;
	Rele9 := FALSE;
	Rele10 := FALSE;
	Rele11 := FALSE;
	Rele12 := TRUE;
END_IF
IF (DlouhyStiskPlus)
THEN
	index := 0;
END_IF

IF (DlouhyStiskMinus)
THEN
	index := 0;
END_IF
END_PROGRAM

(* POU Kolotoc/KolotocF, CFC *)
FUNCTION_BLOCK KolotocF
VAR
END_VAR
VAR_INPUT
	xPlus: BOOL;
	xMinus: BOOL;
	iPocetVystupu: INT;
END_VAR
VAR_OUTPUT
	xOut1: BOOL;
	xOut2: BOOL;
	xOut3: BOOL;
	xOut4: BOOL;
	xOut5: BOOL;
	xOut6: BOOL;
	xOut7: BOOL;
	xOut8: BOOL;
	xOut9: BOOL;
	xOut10: BOOL;
	xOut11: BOOL;
	xOut12: BOOL;
END_VAR
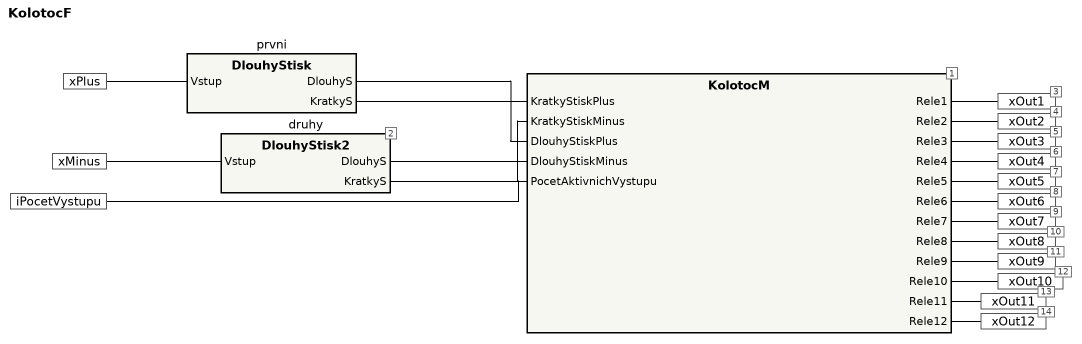
_CFC_ (* Continuous Function Chart, elements in execution order *)
#0 prvni:DlouhyStisk(Vstup: xPlus)
#1 KolotocM(KratkyStiskPlus: #0.KratkyS, KratkyStiskMinus: #2.KratkyS, DlouhyStiskPlus: #0.DlouhyS, DlouhyStiskMinus: #2.DlouhyS, PocetAktivnichVystupu: iPocetVystupu)
#2 druhy:DlouhyStisk2(Vstup: xMinus)
#3 xOut1 <= #1.Rele1
#4 xOut2 <= #1.Rele2
#5 xOut3 <= #1.Rele3
#6 xOut4 <= #1.Rele4
#7 xOut5 <= #1.Rele5
#8 xOut6 <= #1.Rele6
#9 xOut7 <= #1.Rele7
#10 xOut8 <= #1.Rele8
#11 xOut9 <= #1.Rele9
#12 xOut10 <= #1.Rele10
#13 xOut11 <= #1.Rele11
#14 xOut12 <= #1.Rele12
_END_CFC_
(* the same logic as Structured Text *)
prvni(Vstup := xPlus);
KolotocM(KratkyStiskPlus := prvni.KratkyS, KratkyStiskMinus := druhy.KratkyS, DlouhyStiskPlus := prvni.DlouhyS, DlouhyStiskMinus := druhy.DlouhyS, PocetAktivnichVystupu := iPocetVystupu);
druhy(Vstup := xMinus);
xOut1 := KolotocM.Rele1;
xOut2 := KolotocM.Rele2;
xOut3 := KolotocM.Rele3;
xOut4 := KolotocM.Rele4;
xOut5 := KolotocM.Rele5;
xOut6 := KolotocM.Rele6;
xOut7 := KolotocM.Rele7;
xOut8 := KolotocM.Rele8;
xOut9 := KolotocM.Rele9;
xOut10 := KolotocM.Rele10;
xOut11 := KolotocM.Rele11;
xOut12 := KolotocM.Rele12;
END_FUNCTION_BLOCK

(* Visualisation Addressing
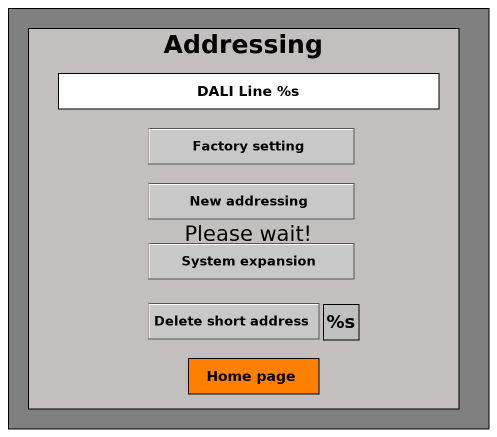
rectangle at (185,80)-(616,461): text "Addressing"
button at (305,235)-(511,271): text "New addressing"; taps DALI_Config.NewAddress; tooltip You have to click and hold the button "New Addressing" longer than two seconds to start the new addressing.
button at (305,295)-(511,331): text "System expansion"; taps DALI_Config.xErweitert; tooltip If you click the button "System expansion", only the ECGs with no short address will be addressed.
rectangle at (480,356)-(516,392): text "%s"; shows DALI_Config.LoeschKurzadr; tooltip Enter the short address to be deleted (1 - 64).; editable
rounded rectangle at (345,410)-(476,446): text "Home page"; opens DALI; tooltip Back to home page
button at (305,180)-(511,216): text "Factory setting"; taps DALI_Config.Reset; tooltip To reset the ECG you have to click and hold the button two seconds. Group and scene configurations will be deleted.
button at (305,355)-(476,391): text "Delete short address"; taps DALI_Config.Loeschen; tooltip The selected short address will be deleted.
rectangle at (265,100)-(546,471): text "Please wait!"; invisible if not DALI_Config.JobMerker[5]
rounded rectangle at (215,125)-(596,161): text "DALI Line %s"; shows DALI_Config.bDali_Linie; tooltip You can change the DALI Line only on the home page.
1 more shapes without text or variables
*)

(* Visualisation CasProg
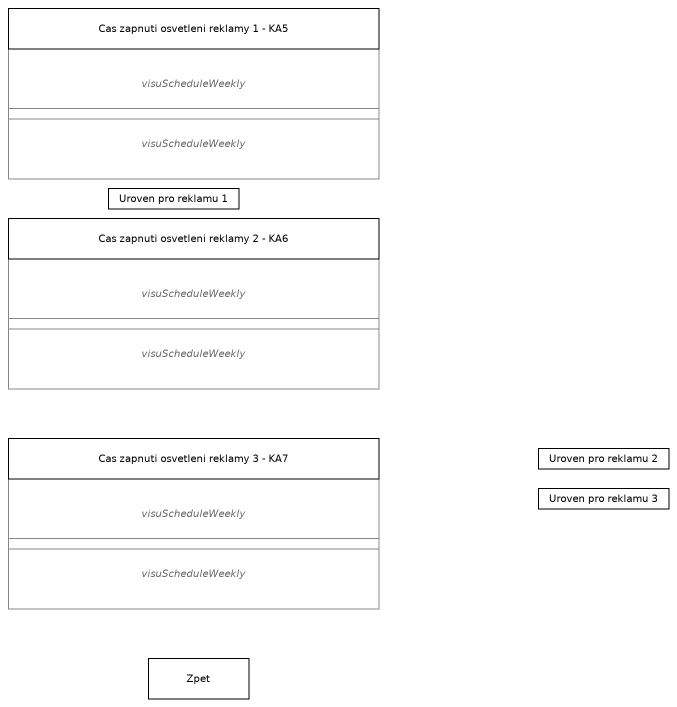
embedded screen at (30,60)-(401,131): visuScheduleWeekly
embedded screen at (30,120)-(401,191): visuScheduleWeekly
rectangle at (30,20)-(401,61): text "Cas zapnuti osvetleni reklamy 1 - KA5"
rectangle at (130,200)-(261,221): text "Uroven pro reklamu 1"
rectangle at (170,670)-(271,711): text "Zpet"; opens ZOOMTOCALLER
embedded screen at (30,270)-(401,341): visuScheduleWeekly
embedded screen at (30,330)-(401,401): visuScheduleWeekly
rectangle at (30,230)-(401,271): text "Cas zapnuti osvetleni reklamy 2 - KA6"
rectangle at (560,460)-(691,481): text "Uroven pro reklamu 2"
embedded screen at (30,490)-(401,561): visuScheduleWeekly
embedded screen at (30,550)-(401,621): visuScheduleWeekly
rectangle at (30,450)-(401,491): text "Cas zapnuti osvetleni reklamy 3 - KA7"
rectangle at (560,500)-(691,521): text "Uroven pro reklamu 3"
3 elements of other kinds (tables, trends, ...) not read
*)

(* Visualisation DALI
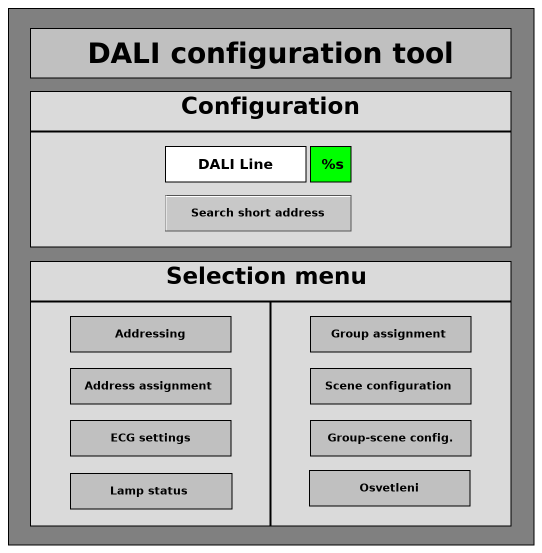
rectangle at (171,91)-(652,247): text "Configuration"
rectangle at (171,261)-(652,526): text "Selection menu"
rectangle at (171,28)-(652,78): text "DALI configuration tool"
rectangle at (211,316)-(372,352): text "Addressing"; opens Addressing
rectangle at (211,368)-(372,404): text "Address assignment"; opens Sort_short_address
rectangle at (451,316)-(612,352): text "Group assignment"; opens group_assignment
rectangle at (451,368)-(612,404): text "Scene configuration"; opens Scene_configuration
rectangle at (211,420)-(372,456): text "ECG settings"; opens ECG_settings
rectangle at (451,420)-(612,456): text "Group-scene config."; opens GroupSceneConfiguration
rectangle at (306,146)-(447,182): text "DALI Line"
button at (306,195)-(492,231): text "Search short address"; taps DALI_Config.SucheKurzadr; tooltip Clicking the button "Search Short Address" will start the search for available short addresses.
rectangle at (451,146)-(492,182): text "%s"; shows DALI_Config.Dali_Linie; alarm colour if DALI_Config.keineJobliste; tooltip Select DALI Line (1 - 5); editable
rectangle at (211,473)-(373,509): text "Lamp status"; opens Lamp_status
rectangle at (450,470)-(611,506): text "Osvetleni"; opens PLC_VISU
4 more shapes without text or variables
*)

(* Visualisation DALI_cfg
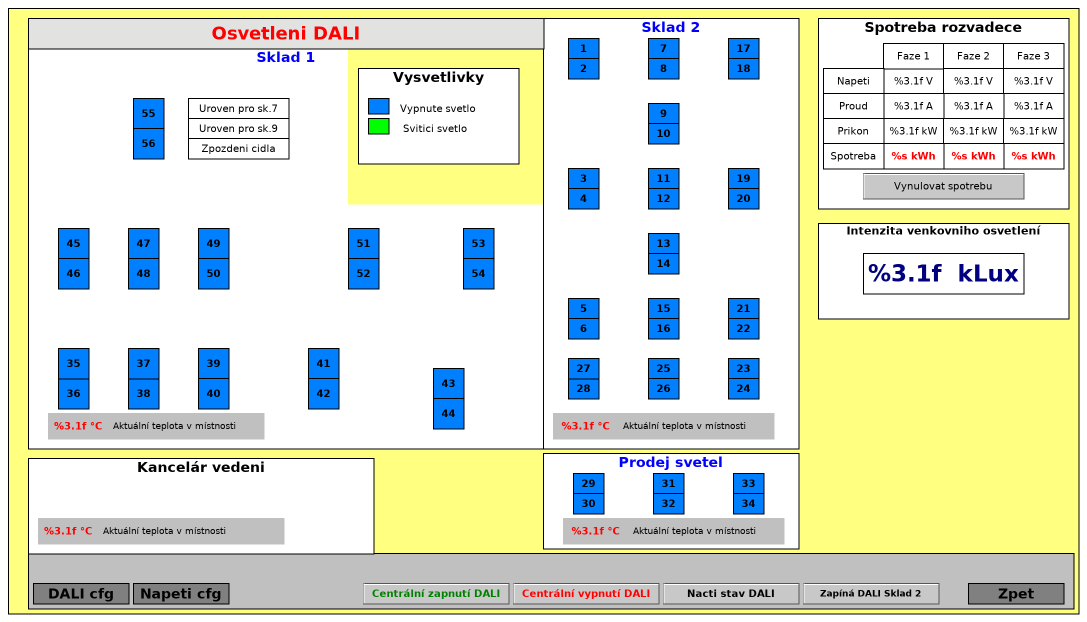
rectangle at (30,50)-(546,451): text "Sklad 1"
rounded rectangle at (360,70)-(521,166): text "Vysvetlivky"
rectangle at (545,455)-(801,551): text "Prodej svetel"; opens prodej_svetel
rectangle at (545,20)-(801,451): text "Sklad 2"; opens prodej_svetel
rectangle at (570,40)-(601,61): text "1"; alarm colour if DALI_Config.Kurzadr[1]
rectangle at (570,40)-(601,61): text "1"; invisible if not DALI_Config.Kurzadr[1]; alarm colour if DALI_Config.LampeEin[1]
rectangle at (570,60)-(601,81): text "2"; alarm colour if DALI_Config.Kurzadr[2]
rectangle at (570,60)-(601,81): text "2"; invisible if not DALI_Config.Kurzadr[2]; alarm colour if DALI_Config.LampeEin[2]
rectangle at (570,170)-(601,191): text "3"; alarm colour if DALI_Config.Kurzadr[3]
rectangle at (570,170)-(601,191): text "3"; invisible if not DALI_Config.Kurzadr[3]; alarm colour if DALI_Config.LampeEin[3]
rectangle at (570,190)-(601,211): text "4"; alarm colour if DALI_Config.Kurzadr[4]
rectangle at (570,190)-(601,211): text "4"; invisible if not DALI_Config.Kurzadr[4]; alarm colour if DALI_Config.LampeEin[4]
rectangle at (570,300)-(601,321): text "5"; alarm colour if DALI_Config.Kurzadr[5]
rectangle at (570,300)-(601,321): text "5"; invisible if not DALI_Config.Kurzadr[5]; alarm colour if DALI_Config.LampeEin[5]
rectangle at (570,320)-(601,341): text "6"; alarm colour if DALI_Config.Kurzadr[6]
rectangle at (570,320)-(601,341): text "6"; invisible if not DALI_Config.Kurzadr[6]; alarm colour if DALI_Config.LampeEin[6]
rectangle at (650,40)-(681,61): text "7"; alarm colour if DALI_Config.Kurzadr[7]
rectangle at (650,40)-(681,61): text "7"; invisible if not DALI_Config.Kurzadr[7]; alarm colour if DALI_Config.LampeEin[7]
rectangle at (650,60)-(681,81): text "8"; alarm colour if DALI_Config.Kurzadr[8]
rectangle at (650,60)-(681,81): text "8"; invisible if not DALI_Config.Kurzadr[8]; alarm colour if DALI_Config.LampeEin[8]
rectangle at (650,105)-(681,126): text "9"; alarm colour if DALI_Config.Kurzadr[9]
rectangle at (650,105)-(681,126): text "9"; invisible if not DALI_Config.Kurzadr[9]; alarm colour if DALI_Config.LampeEin[9]
rectangle at (650,125)-(681,146): text "10"; alarm colour if DALI_Config.Kurzadr[10]
rectangle at (650,125)-(681,146): text "10"; invisible if not DALI_Config.Kurzadr[10]; alarm colour if DALI_Config.LampeEin[10]
rectangle at (650,170)-(681,191): text "11"; alarm colour if DALI_Config.Kurzadr[11]
rectangle at (650,170)-(681,191): text "11"; invisible if not DALI_Config.Kurzadr[11]; alarm colour if DALI_Config.LampeEin[11]
rectangle at (650,190)-(681,211): text "12"; alarm colour if DALI_Config.Kurzadr[12]
rectangle at (650,190)-(681,211): text "12"; invisible if not DALI_Config.Kurzadr[12]; alarm colour if DALI_Config.LampeEin[12]
rectangle at (650,235)-(681,256): text "13"; alarm colour if DALI_Config.Kurzadr[13]
rectangle at (650,235)-(681,256): text "13"; invisible if not DALI_Config.Kurzadr[13]; alarm colour if DALI_Config.LampeEin[13]
rectangle at (650,255)-(681,276): text "14"; alarm colour if DALI_Config.Kurzadr[14]
rectangle at (650,255)-(681,276): text "14"; invisible if not DALI_Config.Kurzadr[14]; alarm colour if DALI_Config.LampeEin[14]
rectangle at (650,300)-(681,321): text "15"; alarm colour if DALI_Config.Kurzadr[15]
rectangle at (650,300)-(681,321): text "15"; invisible if not DALI_Config.Kurzadr[15]; alarm colour if DALI_Config.LampeEin[15]
rectangle at (650,320)-(681,341): text "16"; alarm colour if DALI_Config.Kurzadr[16]
rectangle at (650,320)-(681,341): text "16"; invisible if not DALI_Config.Kurzadr[16]; alarm colour if DALI_Config.LampeEin[16]
rectangle at (730,40)-(761,61): text "17"; alarm colour if DALI_Config.Kurzadr[17]
rectangle at (730,40)-(761,61): text "17"; invisible if not DALI_Config.Kurzadr[17]; alarm colour if DALI_Config.LampeEin[17]
rectangle at (730,170)-(761,191): text "19"; alarm colour if DALI_Config.Kurzadr[19]
rectangle at (730,170)-(761,191): text "19"; invisible if not DALI_Config.Kurzadr[19]; alarm colour if DALI_Config.LampeEin[19]
rectangle at (730,60)-(761,81): text "18"; alarm colour if DALI_Config.Kurzadr[18]
rectangle at (730,60)-(761,81): text "18"; invisible if not DALI_Config.Kurzadr[18]; alarm colour if DALI_Config.LampeEin[18]
rectangle at (730,190)-(761,211): text "20"; alarm colour if DALI_Config.Kurzadr[20]
rectangle at (730,190)-(761,211): text "20"; invisible if not DALI_Config.Kurzadr[20]; alarm colour if DALI_Config.LampeEin[20]
rectangle at (730,300)-(761,321): text "21"; alarm colour if DALI_Config.Kurzadr[21]
rectangle at (730,300)-(761,321): text "21"; invisible if not DALI_Config.Kurzadr[21]; alarm colour if DALI_Config.LampeEin[21]
rectangle at (730,320)-(761,341): text "22"; alarm colour if DALI_Config.Kurzadr[22]
rectangle at (730,320)-(761,341): text "22"; invisible if not DALI_Config.Kurzadr[22]; alarm colour if DALI_Config.LampeEin[22]
rectangle at (730,360)-(761,381): text "23"; alarm colour if DALI_Config.Kurzadr[23]
rectangle at (730,360)-(761,381): text "23"; invisible if not DALI_Config.Kurzadr[23]; alarm colour if DALI_Config.LampeEin[23]
rectangle at (730,380)-(761,401): text "24"; alarm colour if DALI_Config.Kurzadr[24]
rectangle at (730,380)-(761,401): text "24"; invisible if not DALI_Config.Kurzadr[24]; alarm colour if DALI_Config.LampeEin[24]
rectangle at (650,360)-(681,381): text "25"; alarm colour if DALI_Config.Kurzadr[25]
rectangle at (650,360)-(681,381): text "25"; invisible if not DALI_Config.Kurzadr[25]; alarm colour if DALI_Config.LampeEin[25]
rectangle at (575,475)-(606,496): text "29"; alarm colour if DALI_Config.Kurzadr[29]
rectangle at (575,475)-(606,496): text "29"; invisible if not DALI_Config.Kurzadr[29]; alarm colour if DALI_Config.LampeEin[29]
rectangle at (570,380)-(601,401): text "28"; alarm colour if DALI_Config.Kurzadr[28]
rectangle at (570,380)-(601,401): text "28"; invisible if not DALI_Config.Kurzadr[28]; alarm colour if DALI_Config.LampeEin[28]
rectangle at (570,360)-(601,381): text "27"; alarm colour if DALI_Config.Kurzadr[27]
rectangle at (570,360)-(601,381): text "27"; invisible if not DALI_Config.Kurzadr[27]; alarm colour if DALI_Config.LampeEin[27]
rectangle at (650,380)-(681,401): text "26"; alarm colour if DALI_Config.Kurzadr[26]
rectangle at (650,380)-(681,401): text "26"; invisible if not DALI_Config.Kurzadr[26]; alarm colour if DALI_Config.LampeEin[26]
rectangle at (575,495)-(606,516): text "30"; alarm colour if DALI_Config.Kurzadr[30]
rectangle at (575,495)-(606,516): text "30"; invisible if not DALI_Config.Kurzadr[30]; alarm colour if DALI_Config.LampeEin[30]
rectangle at (655,475)-(686,496): text "31"; alarm colour if DALI_Config.Kurzadr[31]
rectangle at (655,475)-(686,496): text "31"; invisible if not DALI_Config.Kurzadr[31]; alarm colour if DALI_Config.LampeEin[31]
rectangle at (655,495)-(686,516): text "32"; alarm colour if DALI_Config.Kurzadr[32]
rectangle at (655,495)-(686,516): text "32"; invisible if not DALI_Config.Kurzadr[32]; alarm colour if DALI_Config.LampeEin[32]
rectangle at (735,475)-(766,496): text "33"; alarm colour if DALI_Config.Kurzadr[33]
rectangle at (735,475)-(766,496): text "33"; invisible if not DALI_Config.Kurzadr[33]; alarm colour if DALI_Config.LampeEin[33]
rectangle at (735,495)-(766,516): text "34"; alarm colour if DALI_Config.Kurzadr[34]
rectangle at (735,495)-(766,516): text "34"; invisible if not DALI_Config.Kurzadr[34]; alarm colour if DALI_Config.LampeEin[34]
rectangle at (60,380)-(91,411): text "36"; alarm colour if DALI_Config.Kurzadr[36]
rectangle at (60,380)-(91,411): text "36"; invisible if not DALI_Config.Kurzadr[36]; alarm colour if DALI_Config.LampeEin[36]
rectangle at (130,380)-(161,411): text "38"; alarm colour if DALI_Config.Kurzadr[38]
rectangle at (130,380)-(161,411): text "38"; invisible if not DALI_Config.Kurzadr[38]; alarm colour if DALI_Config.LampeEin[38]
rectangle at (200,350)-(231,381): text "39"; alarm colour if DALI_Config.Kurzadr[39]
rectangle at (200,350)-(231,381): text "39"; invisible if not DALI_Config.Kurzadr[39]; alarm colour if DALI_Config.LampeEin[39]
rectangle at (130,350)-(161,381): text "37"; alarm colour if DALI_Config.Kurzadr[37]
rectangle at (130,350)-(161,381): text "37"; invisible if not DALI_Config.Kurzadr[37]; alarm colour if DALI_Config.LampeEin[37]
rectangle at (60,350)-(91,381): text "35"; alarm colour if DALI_Config.Kurzadr[35]
rectangle at (60,350)-(91,381): text "35"; invisible if not DALI_Config.Kurzadr[35]; alarm colour if DALI_Config.LampeEin[35]
rectangle at (310,350)-(341,381): text "41"; alarm colour if DALI_Config.Kurzadr[41]
rectangle at (310,350)-(341,381): text "41"; invisible if not DALI_Config.Kurzadr[41]; alarm colour if DALI_Config.LampeEin[41]
rectangle at (310,380)-(341,411): text "42"; alarm colour if DALI_Config.Kurzadr[42]
rectangle at (310,380)-(341,411): text "42"; invisible if not DALI_Config.Kurzadr[42]; alarm colour if DALI_Config.LampeEin[42]
rectangle at (200,380)-(231,411): text "40"; alarm colour if DALI_Config.Kurzadr[40]
rectangle at (200,380)-(231,411): text "40"; invisible if not DALI_Config.Kurzadr[40]; alarm colour if DALI_Config.LampeEin[40]
rectangle at (435,370)-(466,401): text "43"; alarm colour if DALI_Config.Kurzadr[43]
rectangle at (435,370)-(466,401): text "43"; invisible if not DALI_Config.Kurzadr[43]; alarm colour if DALI_Config.LampeEin[43]
rectangle at (435,400)-(466,431): text "44"; alarm colour if DALI_Config.Kurzadr[44]
rectangle at (435,400)-(466,431): text "44"; invisible if not DALI_Config.Kurzadr[44]; alarm colour if DALI_Config.LampeEin[44]
rectangle at (60,230)-(91,261): text "45"; alarm colour if DALI_Config.Kurzadr[45]
rectangle at (60,230)-(91,261): text "45"; invisible if not DALI_Config.Kurzadr[45]; alarm colour if DALI_Config.LampeEin[45]
rectangle at (60,260)-(91,291): text "46"; alarm colour if DALI_Config.Kurzadr[46]
rectangle at (60,260)-(91,291): text "46"; invisible if not DALI_Config.Kurzadr[46]; alarm colour if DALI_Config.LampeEin[46]
rectangle at (130,230)-(161,261): text "47"; alarm colour if DALI_Config.Kurzadr[47]
rectangle at (130,230)-(161,261): text "47"; invisible if not DALI_Config.Kurzadr[47]; alarm colour if DALI_Config.LampeEin[47]
rectangle at (130,260)-(161,291): text "48"; alarm colour if DALI_Config.Kurzadr[48]
rectangle at (130,260)-(161,291): text "48"; invisible if not DALI_Config.Kurzadr[48]; alarm colour if DALI_Config.LampeEin[48]
rectangle at (200,230)-(231,261): text "49"; alarm colour if DALI_Config.Kurzadr[49]
rectangle at (200,230)-(231,261): text "49"; invisible if not DALI_Config.Kurzadr[49]; alarm colour if DALI_Config.LampeEin[49]
rectangle at (200,260)-(231,291): text "50"; alarm colour if DALI_Config.Kurzadr[50]
rectangle at (200,260)-(231,291): text "50"; invisible if not DALI_Config.Kurzadr[50]; alarm colour if DALI_Config.LampeEin[50]
rectangle at (350,230)-(381,261): text "51"; alarm colour if DALI_Config.Kurzadr[51]
rectangle at (350,230)-(381,261): text "51"; invisible if not DALI_Config.Kurzadr[51]; alarm colour if DALI_Config.LampeEin[51]
rectangle at (350,260)-(381,291): text "52"; alarm colour if DALI_Config.Kurzadr[52]
rectangle at (350,260)-(381,291): text "52"; invisible if not DALI_Config.Kurzadr[52]; alarm colour if DALI_Config.LampeEin[52]
rectangle at (465,230)-(496,261): text "53"; alarm colour if DALI_Config.Kurzadr[53]
rectangle at (465,230)-(496,261): text "53"; invisible if not DALI_Config.Kurzadr[53]; alarm colour if DALI_Config.LampeEin[53]
rectangle at (465,260)-(496,291): text "54"; alarm colour if DALI_Config.Kurzadr[54]
rectangle at (465,260)-(496,291): text "54"; invisible if not DALI_Config.Kurzadr[54]; alarm colour if DALI_Config.LampeEin[54]
rectangle at (135,100)-(166,131): text "55"; alarm colour if DALI_Config.Kurzadr[55]
rectangle at (135,100)-(166,131): text "55"; invisible if not DALI_Config.Kurzadr[55]; alarm colour if DALI_Config.LampeEin[55]
rectangle at (135,130)-(166,161): text "56"; alarm colour if DALI_Config.Kurzadr[56]
rectangle at (135,130)-(166,161): text "56"; invisible if not DALI_Config.Kurzadr[56]; alarm colour if DALI_Config.LampeEin[56]
rectangle at (30,20)-(546,51): text "Osvetleni DALI"
button at (665,585)-(801,606): text "Nacti stav DALI"; taps DALI_Config.Status; tooltip Kliknutim nactete status svetel. (sviti, nesviti, vadna).
rectangle at (400,100)-(516,121): text "Vypnute svetlo"
rectangle at (400,120)-(536,141): text "Svitici svetlo"
rectangle at (565,520)-(631,546): text "%3.1f °C"; shows .Teplota_2/10.0
rectangle at (630,520)-(786,546): text "Aktuální teplota v místnosti"
rectangle at (620,415)-(776,441): text "Aktuální teplota v místnosti"
rectangle at (110,415)-(266,441): text "Aktuální teplota v místnosti"
rectangle at (555,415)-(621,441): text "%3.1f °C"; shows .Teplota_1/10.0
rectangle at (50,415)-(111,441): text "%3.1f °C"; shows .Teplota_3/10.0
button at (365,585)-(511,606): text "Centrální zapnutí DALI"; taps DALI_Config.Ein; tooltip Vsechny DALI svetla zapni
button at (515,585)-(661,606): text "Centrální vypnutí DALI"; taps DALI_Config.Aus; tooltip Vsechny DALI svetla vypni
rounded rectangle at (820,20)-(1071,211): text "Spotreba rozvadece"
rectangle at (885,70)-(946,96): text "%3.1f V"; shows TriFaze.arNapeti[1]
rectangle at (885,45)-(946,71): text "Faze 1"
rectangle at (945,45)-(1006,71): text "Faze 2"
rectangle at (1005,45)-(1066,71): text "Faze 3"
rectangle at (945,70)-(1006,96): text "%3.1f V"; shows TriFaze.arNapeti[2]
rectangle at (1005,70)-(1066,96): text "%3.1f V"; shows TriFaze.arNapeti[3]
rectangle at (1005,95)-(1066,121): text "%3.1f A"; shows TriFaze.arProud[3]
rectangle at (945,95)-(1006,121): text "%3.1f A"; shows TriFaze.arProud[2]
rectangle at (885,95)-(946,121): text "%3.1f A"; shows TriFaze.arProud[1]
rectangle at (885,120)-(946,146): text "%3.1f kW"; shows TriFaze.arVykon[1]
rectangle at (945,120)-(1006,146): text "%3.1f kW"; shows TriFaze.arVykon[2]
rectangle at (1005,120)-(1066,146): text "%3.1f kW"; shows TriFaze.arVykon[3]
rectangle at (1005,145)-(1066,171): text "%s kWh"; shows TriFaze.adwSpotreba[3]
rectangle at (945,145)-(1006,171): text "%s kWh"; shows TriFaze.adwSpotreba[2]
rectangle at (885,145)-(946,171): text "%s kWh"; shows TriFaze.adwSpotreba[1]
button at (865,175)-(1026,201): text "Vynulovat spotrebu"; taps TriFaze.SmazL1
rounded rectangle at (820,225)-(1071,321): text "Intenzita venkovniho osvetlení"; opens lux
rectangle at (865,255)-(1026,296): text "%3.1f  kLux"; shows .Analog_1/3276.4*2
rectangle at (825,70)-(886,96): text "Napeti"
rectangle at (825,95)-(886,121): text "Proud"
rectangle at (825,120)-(886,146): text "Prikon"
rectangle at (825,145)-(886,171): text "Spotreba"
rectangle at (30,460)-(376,556): text "Kancelár vedeni"
rectangle at (100,520)-(286,546): text "Aktuální teplota v místnosti"
rectangle at (40,520)-(101,546): text "%3.1f °C"; shows .Teplota_4/10.0
rectangle at (970,585)-(1066,606): text "Zpet"; opens PLC_VISU; tooltip Na úvodní stranu
rectangle at (135,585)-(231,606): text "Napeti cfg"; opens Visualizace; tooltip Back to home page
button at (805,585)-(941,606): text "Zapíná DALI Sklad 2"; taps .TL01s; tooltip 1x zapne/vypne, 2x zapne skupinu 2, 3x zapne vše
rectangle at (35,585)-(131,606): text "DALI cfg"; opens DALI; tooltip Back to home page
rectangle at (190,100)-(291,121): text "Uroven pro sk.7"
rectangle at (190,120)-(291,141): text "Uroven pro sk.9"
rectangle at (190,140)-(291,161): text "Zpozdeni cidla"
6 more shapes without text or variables
3 elements of other kinds (tables, trends, ...) not read
*)

(* Visualisation ECG_settings
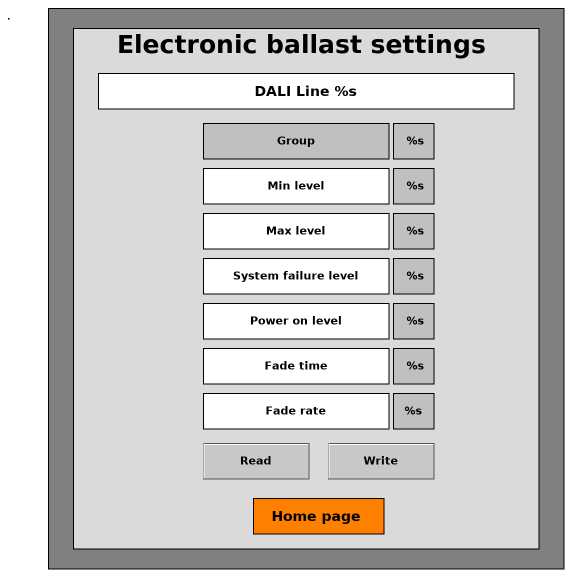
rectangle at (150,40)-(616,561): text "Electronic ballast settings"
rectangle at (280,225)-(466,261): text "Max level"
rectangle at (280,180)-(466,216): text "Min level"
rectangle at (280,270)-(466,306): text "System failure level"
rectangle at (280,315)-(466,351): text "Power on level"
rectangle at (280,360)-(466,396): text "Fade time"
rectangle at (280,405)-(466,441): text "Fade rate"
rectangle at (280,135)-(466,171): text "Short address"; invisible if DALI_Config.Kurzadr_Gruppe; toggles DALI_Config.Kurzadr_Gruppe
rectangle at (280,135)-(466,171): text "Group"; invisible if not DALI_Config.Kurzadr_Gruppe; toggles DALI_Config.Kurzadr_Gruppe; tooltip Selection group or short address
rectangle at (470,135)-(511,171): text "%s"; shows DALI_Config.Adresse; tooltip Enter group (1-16) or short address (1 - 64); editable
rounded rectangle at (330,510)-(461,546): text "Home page"; opens DALI; tooltip Back to home page
rectangle at (470,180)-(511,216): text "%s"; shows DALI_Config.MinLevel; tooltip Minimal brightness level in percent. Min level has to be smaller than max level.; editable
rectangle at (470,225)-(511,261): text "%s"; shows DALI_Config.MaxLevel; tooltip Maximum brightness level in percent; editable
rectangle at (470,270)-(511,306): text "%s"; shows DALI_Config.SystemFailure; tooltip Brightness level in percent in case of a system failure. The value 101 means "MASK".; editable
rectangle at (470,315)-(511,351): text "%s"; shows DALI_Config.PowerOn; tooltip Brightness level in percent if the ECGs are powered on.; editable
rectangle at (470,360)-(511,396): text "%s"; shows DALI_Config.Konfig[4]; tooltip Enter the fade time (0 - 15); editable
rectangle at (470,405)-(511,441): text "%s"; shows DALI_Config.Konfig[5]; tooltip Enter the fade rate (1 -15); editable
button at (280,455)-(386,491): text "Read"; taps DALI_Config.Lese; tooltip If you click the button "Read", the settings of the ECG will be read. Group queries are not possible.
button at (405,455)-(511,491): text "Write"; taps DALI_Config.Schreib; tooltip If you click the button "Write", the new settings will be written into the ECG.
rounded rectangle at (175,85)-(591,121): text "DALI Line %s"; shows DALI_Config.bDali_Linie; tooltip You can change the DALI Line only on the home page.
2 more shapes without text or variables
*)

(* Visualisation Group_assignment
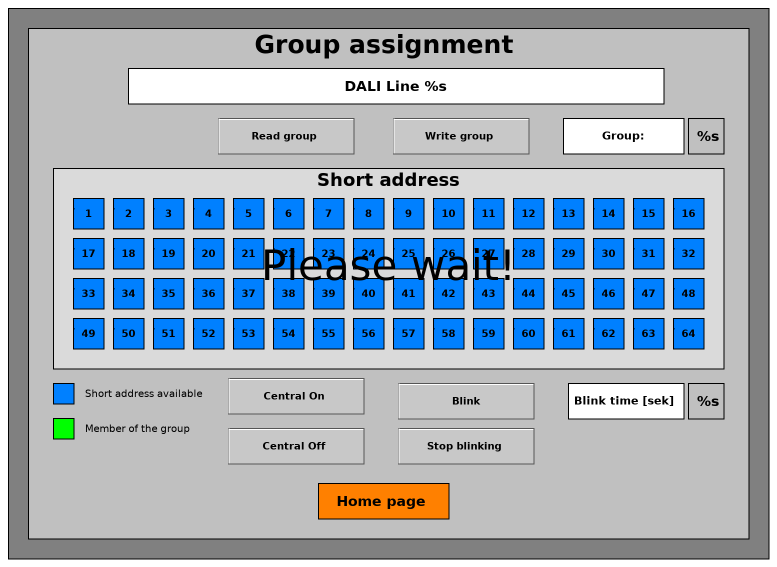
rectangle at (40,40)-(761,551): text "Group assignment"
rounded rectangle at (330,495)-(461,531): text "Home page"; opens DALI; tooltip Back to home page
rectangle at (65,180)-(736,381): text "Short address"
rectangle at (85,210)-(116,241): text "1"; alarm colour if DALI_Config.Kurzadr[1]
rectangle at (85,210)-(116,241): text "1"; invisible if not DALI_Config.Kurzadr[1]; alarm colour if DALI_Config.Gruppenadr[1]; toggles DALI_Config.Gruppenadr[1]
rectangle at (125,210)-(156,241): text "2"; alarm colour if DALI_Config.Kurzadr[2]
rectangle at (125,210)-(156,241): text "2"; invisible if not DALI_Config.Kurzadr[2]; alarm colour if DALI_Config.Gruppenadr[2]; toggles DALI_Config.Gruppenadr[2]
rectangle at (165,210)-(196,241): text "3"; alarm colour if DALI_Config.Kurzadr[3]
rectangle at (165,210)-(196,241): text "3"; invisible if not DALI_Config.Kurzadr[3]; alarm colour if DALI_Config.Gruppenadr[3]; toggles DALI_Config.Gruppenadr[3]
rectangle at (205,210)-(236,241): text "4"; alarm colour if DALI_Config.Kurzadr[4]
rectangle at (205,210)-(236,241): text "4"; invisible if not DALI_Config.Kurzadr[4]; alarm colour if DALI_Config.Gruppenadr[4]; toggles DALI_Config.Gruppenadr[4]
rectangle at (245,210)-(276,241): text "5"; alarm colour if DALI_Config.Kurzadr[5]
rectangle at (245,210)-(276,241): text "5"; invisible if not DALI_Config.Kurzadr[5]; alarm colour if DALI_Config.Gruppenadr[5]; toggles DALI_Config.Gruppenadr[5]
rectangle at (285,210)-(316,241): text "6"; alarm colour if DALI_Config.Kurzadr[6]
rectangle at (285,210)-(316,241): text "6"; invisible if not DALI_Config.Kurzadr[6]; alarm colour if DALI_Config.Gruppenadr[6]; toggles DALI_Config.Gruppenadr[6]
rectangle at (325,210)-(356,241): text "7"; alarm colour if DALI_Config.Kurzadr[7]
rectangle at (325,210)-(356,241): text "7"; invisible if not DALI_Config.Kurzadr[7]; alarm colour if DALI_Config.Gruppenadr[7]; toggles DALI_Config.Gruppenadr[7]
rectangle at (365,210)-(396,241): text "8"; alarm colour if DALI_Config.Kurzadr[8]
rectangle at (365,210)-(396,241): text "8"; invisible if not DALI_Config.Kurzadr[8]; alarm colour if DALI_Config.Gruppenadr[8]; toggles DALI_Config.Gruppenadr[8]
rectangle at (405,210)-(436,241): text "9"; alarm colour if DALI_Config.Kurzadr[9]
rectangle at (405,210)-(436,241): text "9"; invisible if not DALI_Config.Kurzadr[9]; alarm colour if DALI_Config.Gruppenadr[9]; toggles DALI_Config.Gruppenadr[9]
rectangle at (445,210)-(476,241): text "10"; alarm colour if DALI_Config.Kurzadr[10]
rectangle at (445,210)-(476,241): text "10"; invisible if not DALI_Config.Kurzadr[10]; alarm colour if DALI_Config.Gruppenadr[10]; toggles DALI_Config.Gruppenadr[10]
rectangle at (485,210)-(516,241): text "11"; alarm colour if DALI_Config.Kurzadr[11]
rectangle at (485,210)-(516,241): text "11"; invisible if not DALI_Config.Kurzadr[11]; alarm colour if DALI_Config.Gruppenadr[11]; toggles DALI_Config.Gruppenadr[11]
rectangle at (525,210)-(556,241): text "12"; alarm colour if DALI_Config.Kurzadr[12]
rectangle at (525,210)-(556,241): text "12"; invisible if not DALI_Config.Kurzadr[12]; alarm colour if DALI_Config.Gruppenadr[12]; toggles DALI_Config.Gruppenadr[12]
rectangle at (565,210)-(596,241): text "13"; alarm colour if DALI_Config.Kurzadr[13]
rectangle at (565,210)-(596,241): text "13"; invisible if not DALI_Config.Kurzadr[13]; alarm colour if DALI_Config.Gruppenadr[13]; toggles DALI_Config.Gruppenadr[13]
rectangle at (605,210)-(636,241): text "14"; alarm colour if DALI_Config.Kurzadr[14]
rectangle at (605,210)-(636,241): text "14"; invisible if not DALI_Config.Kurzadr[14]; alarm colour if DALI_Config.Gruppenadr[14]; toggles DALI_Config.Gruppenadr[14]
rectangle at (645,210)-(676,241): text "15"; alarm colour if DALI_Config.Kurzadr[15]
rectangle at (645,210)-(676,241): text "15"; invisible if not DALI_Config.Kurzadr[15]; alarm colour if DALI_Config.Gruppenadr[15]; toggles DALI_Config.Gruppenadr[15]
rectangle at (685,210)-(716,241): text "16"; alarm colour if DALI_Config.Kurzadr[16]
rectangle at (685,210)-(716,241): text "16"; invisible if not DALI_Config.Kurzadr[16]; alarm colour if DALI_Config.Gruppenadr[16]; toggles DALI_Config.Gruppenadr[16]
button at (405,130)-(541,166): text "Write group"; taps DALI_Config.Gruppenkonfiguration; tooltip If you click the button "Write Group", the marked short addresses will be saved as a group.
rectangle at (575,130)-(696,166): text "Group:"
rectangle at (700,130)-(736,166): text "%s"; shows DALI_Config.Gruppe; tooltip Enter the number of the group (1 - 16); editable
button at (410,395)-(546,431): text "Blink"; taps DALI_Config.BlinkenGruppe; tooltip If you click the button "Blink", the selected ECG will blink as long as defined by the "Blink Time" parameter.
button at (410,440)-(546,476): text "Stop blinking"; taps DALI_Config.xBlinken_Aus; tooltip If you click the button "Stop blinking", the blinking of the ECG will stop immediately.
button at (230,130)-(366,166): text "Read group"; taps DALI_Config.GruppeLesen; tooltip If you click the button "Read Group", the short addresses that belong to the group will be displayed.
rectangle at (95,395)-(226,416): text "Short address available"
rectangle at (95,430)-(246,451): text "Member of the group"
rounded rectangle at (140,80)-(676,116): text "DALI Line %s"; shows DALI_Config.bDali_Linie; tooltip You can change the DALI Line only on the home page.
rectangle at (85,250)-(116,281): text "17"; alarm colour if DALI_Config.Kurzadr[17]
rectangle at (85,250)-(116,281): text "17"; invisible if not DALI_Config.Kurzadr[17]; alarm colour if DALI_Config.Gruppenadr[17]; toggles DALI_Config.Gruppenadr[17]
rectangle at (125,250)-(156,281): text "18"; alarm colour if DALI_Config.Kurzadr[18]
rectangle at (125,250)-(156,281): text "18"; invisible if not DALI_Config.Kurzadr[18]; alarm colour if DALI_Config.Gruppenadr[18]; toggles DALI_Config.Gruppenadr[18]
rectangle at (165,250)-(196,281): text "19"; alarm colour if DALI_Config.Kurzadr[19]
rectangle at (165,250)-(196,281): text "19"; invisible if not DALI_Config.Kurzadr[19]; alarm colour if DALI_Config.Gruppenadr[19]; toggles DALI_Config.Gruppenadr[19]
rectangle at (205,250)-(236,281): text "20"; alarm colour if DALI_Config.Kurzadr[20]
rectangle at (205,250)-(236,281): text "20"; invisible if not DALI_Config.Kurzadr[20]; alarm colour if DALI_Config.Gruppenadr[20]; toggles DALI_Config.Gruppenadr[20]
rectangle at (245,250)-(276,281): text "21"; alarm colour if DALI_Config.Kurzadr[21]
rectangle at (245,250)-(276,281): text "21"; invisible if not DALI_Config.Kurzadr[21]; alarm colour if DALI_Config.Gruppenadr[21]; toggles DALI_Config.Gruppenadr[21]
rectangle at (285,250)-(316,281): text "22"; alarm colour if DALI_Config.Kurzadr[22]
rectangle at (285,250)-(316,281): text "22"; invisible if not DALI_Config.Kurzadr[22]; alarm colour if DALI_Config.Gruppenadr[22]; toggles DALI_Config.Gruppenadr[22]
rectangle at (325,250)-(356,281): text "23"; alarm colour if DALI_Config.Kurzadr[23]
rectangle at (325,250)-(356,281): text "23"; invisible if not DALI_Config.Kurzadr[23]; alarm colour if DALI_Config.Gruppenadr[23]; toggles DALI_Config.Gruppenadr[23]
rectangle at (365,250)-(396,281): text "24"; alarm colour if DALI_Config.Kurzadr[24]
rectangle at (365,250)-(396,281): text "24"; invisible if not DALI_Config.Kurzadr[24]; alarm colour if DALI_Config.Gruppenadr[24]; toggles DALI_Config.Gruppenadr[24]
rectangle at (405,250)-(436,281): text "25"; alarm colour if DALI_Config.Kurzadr[25]
rectangle at (405,250)-(436,281): text "25"; invisible if not DALI_Config.Kurzadr[25]; alarm colour if DALI_Config.Gruppenadr[25]; toggles DALI_Config.Gruppenadr[25]
rectangle at (445,250)-(476,281): text "26"; alarm colour if DALI_Config.Kurzadr[26]
rectangle at (445,250)-(476,281): text "26"; invisible if not DALI_Config.Kurzadr[26]; alarm colour if DALI_Config.Gruppenadr[26]; toggles DALI_Config.Gruppenadr[26]
rectangle at (485,250)-(516,281): text "27"; alarm colour if DALI_Config.Kurzadr[27]
rectangle at (485,250)-(516,281): text "27"; invisible if not DALI_Config.Kurzadr[27]; alarm colour if DALI_Config.Gruppenadr[27]; toggles DALI_Config.Gruppenadr[27]
rectangle at (525,250)-(556,281): text "28"; alarm colour if DALI_Config.Kurzadr[28]
rectangle at (525,250)-(556,281): text "28"; invisible if not DALI_Config.Kurzadr[28]; alarm colour if DALI_Config.Gruppenadr[28]; toggles DALI_Config.Gruppenadr[28]
rectangle at (565,250)-(596,281): text "29"; alarm colour if DALI_Config.Kurzadr[29]
rectangle at (565,250)-(596,281): text "29"; invisible if not DALI_Config.Kurzadr[29]; alarm colour if DALI_Config.Gruppenadr[29]; toggles DALI_Config.Gruppenadr[29]
rectangle at (605,250)-(636,281): text "30"; alarm colour if DALI_Config.Kurzadr[30]
rectangle at (605,250)-(636,281): text "30"; invisible if not DALI_Config.Kurzadr[30]; alarm colour if DALI_Config.Gruppenadr[30]; toggles DALI_Config.Gruppenadr[30]
rectangle at (645,250)-(676,281): text "31"; alarm colour if DALI_Config.Kurzadr[31]
rectangle at (645,250)-(676,281): text "31"; invisible if not DALI_Config.Kurzadr[31]; alarm colour if DALI_Config.Gruppenadr[31]; toggles DALI_Config.Gruppenadr[31]
rectangle at (685,250)-(716,281): text "32"; alarm colour if DALI_Config.Kurzadr[32]
rectangle at (685,250)-(716,281): text "32"; invisible if not DALI_Config.Kurzadr[32]; alarm colour if DALI_Config.Gruppenadr[32]; toggles DALI_Config.Gruppenadr[32]
rectangle at (85,290)-(116,321): text "33"; alarm colour if DALI_Config.Kurzadr[33]
rectangle at (85,290)-(116,321): text "33"; invisible if not DALI_Config.Kurzadr[33]; alarm colour if DALI_Config.Gruppenadr[33]; toggles DALI_Config.Gruppenadr[33]
rectangle at (125,290)-(156,321): text "34"; alarm colour if DALI_Config.Kurzadr[34]
rectangle at (125,290)-(156,321): text "34"; invisible if not DALI_Config.Kurzadr[34]; alarm colour if DALI_Config.Gruppenadr[34]; toggles DALI_Config.Gruppenadr[34]
rectangle at (165,290)-(196,321): text "35"; alarm colour if DALI_Config.Kurzadr[35]
rectangle at (165,290)-(196,321): text "35"; invisible if not DALI_Config.Kurzadr[35]; alarm colour if DALI_Config.Gruppenadr[35]; toggles DALI_Config.Gruppenadr[35]
rectangle at (205,290)-(236,321): text "36"; alarm colour if DALI_Config.Kurzadr[36]
rectangle at (205,290)-(236,321): text "36"; invisible if not DALI_Config.Kurzadr[36]; alarm colour if DALI_Config.Gruppenadr[36]; toggles DALI_Config.Gruppenadr[36]
rectangle at (245,290)-(276,321): text "37"; alarm colour if DALI_Config.Kurzadr[37]
rectangle at (245,290)-(276,321): text "37"; invisible if not DALI_Config.Kurzadr[37]; alarm colour if DALI_Config.Gruppenadr[37]; toggles DALI_Config.Gruppenadr[37]
rectangle at (285,290)-(316,321): text "38"; alarm colour if DALI_Config.Kurzadr[38]
rectangle at (285,290)-(316,321): text "38"; invisible if not DALI_Config.Kurzadr[38]; alarm colour if DALI_Config.Gruppenadr[38]; toggles DALI_Config.Gruppenadr[38]
rectangle at (325,290)-(356,321): text "39"; alarm colour if DALI_Config.Kurzadr[39]
rectangle at (325,290)-(356,321): text "39"; invisible if not DALI_Config.Kurzadr[39]; alarm colour if DALI_Config.Gruppenadr[39]; toggles DALI_Config.Gruppenadr[39]
rectangle at (365,290)-(396,321): text "40"; alarm colour if DALI_Config.Kurzadr[40]
rectangle at (365,290)-(396,321): text "40"; invisible if not DALI_Config.Kurzadr[40]; alarm colour if DALI_Config.Gruppenadr[40]; toggles DALI_Config.Gruppenadr[40]
rectangle at (405,290)-(436,321): text "41"; alarm colour if DALI_Config.Kurzadr[41]
rectangle at (405,290)-(436,321): text "41"; invisible if not DALI_Config.Kurzadr[41]; alarm colour if DALI_Config.Gruppenadr[41]; toggles DALI_Config.Gruppenadr[41]
rectangle at (445,290)-(476,321): text "42"; alarm colour if DALI_Config.Kurzadr[42]
rectangle at (445,290)-(476,321): text "42"; invisible if not DALI_Config.Kurzadr[42]; alarm colour if DALI_Config.Gruppenadr[42]; toggles DALI_Config.Gruppenadr[42]
rectangle at (485,290)-(516,321): text "43"; alarm colour if DALI_Config.Kurzadr[43]
rectangle at (485,290)-(516,321): text "43"; invisible if not DALI_Config.Kurzadr[43]; alarm colour if DALI_Config.Gruppenadr[43]; toggles DALI_Config.Gruppenadr[43]
rectangle at (525,290)-(556,321): text "44"; alarm colour if DALI_Config.Kurzadr[44]
rectangle at (525,290)-(556,321): text "44"; invisible if not DALI_Config.Kurzadr[44]; alarm colour if DALI_Config.Gruppenadr[44]; toggles DALI_Config.Gruppenadr[44]
rectangle at (565,290)-(596,321): text "45"; alarm colour if DALI_Config.Kurzadr[45]
rectangle at (565,290)-(596,321): text "45"; invisible if not DALI_Config.Kurzadr[45]; alarm colour if DALI_Config.Gruppenadr[45]; toggles DALI_Config.Gruppenadr[45]
rectangle at (605,290)-(636,321): text "46"; alarm colour if DALI_Config.Kurzadr[46]
rectangle at (605,290)-(636,321): text "46"; invisible if not DALI_Config.Kurzadr[46]; alarm colour if DALI_Config.Gruppenadr[46]; toggles DALI_Config.Gruppenadr[46]
rectangle at (645,290)-(676,321): text "47"; alarm colour if DALI_Config.Kurzadr[47]
rectangle at (645,290)-(676,321): text "47"; invisible if not DALI_Config.Kurzadr[47]; alarm colour if DALI_Config.Gruppenadr[47]; toggles DALI_Config.Gruppenadr[47]
rectangle at (685,290)-(716,321): text "48"; alarm colour if DALI_Config.Kurzadr[48]
rectangle at (685,290)-(716,321): text "48"; invisible if not DALI_Config.Kurzadr[48]; alarm colour if DALI_Config.Gruppenadr[48]; toggles DALI_Config.Gruppenadr[48]
rectangle at (85,330)-(116,361): text "49"; alarm colour if DALI_Config.Kurzadr[49]
rectangle at (85,330)-(116,361): text "49"; invisible if not DALI_Config.Kurzadr[49]; alarm colour if DALI_Config.Gruppenadr[49]; toggles DALI_Config.Gruppenadr[49]
rectangle at (125,330)-(156,361): text "50"; alarm colour if DALI_Config.Kurzadr[50]
rectangle at (125,330)-(156,361): text "50"; invisible if not DALI_Config.Kurzadr[50]; alarm colour if DALI_Config.Gruppenadr[50]; toggles DALI_Config.Gruppenadr[50]
rectangle at (165,330)-(196,361): text "51"; alarm colour if DALI_Config.Kurzadr[51]
rectangle at (165,330)-(196,361): text "51"; invisible if not DALI_Config.Kurzadr[51]; alarm colour if DALI_Config.Gruppenadr[51]; toggles DALI_Config.Gruppenadr[51]
rectangle at (205,330)-(236,361): text "52"; alarm colour if DALI_Config.Kurzadr[52]
rectangle at (205,330)-(236,361): text "52"; invisible if not DALI_Config.Kurzadr[52]; alarm colour if DALI_Config.Gruppenadr[52]; toggles DALI_Config.Gruppenadr[52]
rectangle at (245,330)-(276,361): text "53"; alarm colour if DALI_Config.Kurzadr[53]
rectangle at (245,330)-(276,361): text "53"; invisible if not DALI_Config.Kurzadr[53]; alarm colour if DALI_Config.Gruppenadr[53]; toggles DALI_Config.Gruppenadr[53]
rectangle at (285,330)-(316,361): text "54"; alarm colour if DALI_Config.Kurzadr[54]
rectangle at (285,330)-(316,361): text "54"; invisible if not DALI_Config.Kurzadr[54]; alarm colour if DALI_Config.Gruppenadr[54]; toggles DALI_Config.Gruppenadr[54]
rectangle at (325,330)-(356,361): text "55"; alarm colour if DALI_Config.Kurzadr[55]
rectangle at (325,330)-(356,361): text "55"; invisible if not DALI_Config.Kurzadr[55]; alarm colour if DALI_Config.Gruppenadr[55]; toggles DALI_Config.Gruppenadr[55]
rectangle at (365,330)-(396,361): text "56"; alarm colour if DALI_Config.Kurzadr[56]
rectangle at (365,330)-(396,361): text "56"; invisible if not DALI_Config.Kurzadr[56]; alarm colour if DALI_Config.Gruppenadr[56]; toggles DALI_Config.Gruppenadr[56]
rectangle at (405,330)-(436,361): text "57"; alarm colour if DALI_Config.Kurzadr[57]
rectangle at (405,330)-(436,361): text "57"; invisible if not DALI_Config.Kurzadr[57]; alarm colour if DALI_Config.Gruppenadr[57]; toggles DALI_Config.Gruppenadr[57]
rectangle at (445,330)-(476,361): text "58"; alarm colour if DALI_Config.Kurzadr[58]
rectangle at (445,330)-(476,361): text "58"; invisible if not DALI_Config.Kurzadr[58]; alarm colour if DALI_Config.Gruppenadr[58]; toggles DALI_Config.Gruppenadr[58]
rectangle at (485,330)-(516,361): text "59"; alarm colour if DALI_Config.Kurzadr[59]
rectangle at (485,330)-(516,361): text "59"; invisible if not DALI_Config.Kurzadr[59]; alarm colour if DALI_Config.Gruppenadr[59]; toggles DALI_Config.Gruppenadr[59]
rectangle at (525,330)-(556,361): text "60"; alarm colour if DALI_Config.Kurzadr[60]
rectangle at (525,330)-(556,361): text "60"; invisible if not DALI_Config.Kurzadr[60]; alarm colour if DALI_Config.Gruppenadr[60]; toggles DALI_Config.Gruppenadr[60]
rectangle at (565,330)-(596,361): text "61"; alarm colour if DALI_Config.Kurzadr[61]
rectangle at (565,330)-(596,361): text "61"; invisible if not DALI_Config.Kurzadr[61]; alarm colour if DALI_Config.Gruppenadr[61]; toggles DALI_Config.Gruppenadr[61]
rectangle at (605,330)-(636,361): text "62"; alarm colour if DALI_Config.Kurzadr[62]
rectangle at (605,330)-(636,361): text "62"; invisible if not DALI_Config.Kurzadr[62]; alarm colour if DALI_Config.Gruppenadr[62]; toggles DALI_Config.Gruppenadr[62]
rectangle at (645,330)-(676,361): text "63"; alarm colour if DALI_Config.Kurzadr[63]
rectangle at (645,330)-(676,361): text "63"; invisible if not DALI_Config.Kurzadr[63]; alarm colour if DALI_Config.Gruppenadr[63]; toggles DALI_Config.Gruppenadr[63]
rectangle at (685,330)-(716,361): text "64"; alarm colour if DALI_Config.Kurzadr[64]
rectangle at (685,330)-(716,361): text "64"; invisible if not DALI_Config.Kurzadr[64]; alarm colour if DALI_Config.Gruppenadr[64]; toggles DALI_Config.Gruppenadr[64]
rectangle at (580,395)-(696,431): text "Blink time [sek]"
button at (240,440)-(376,476): text "Central Off"; taps DALI_Config.Aus; tooltip If you click the button "Central Off", all lamps in the network will be switched off.
button at (240,390)-(376,426): text "Central On"; taps DALI_Config.Ein; tooltip If you click the button "Central On", all lamps in the network will be switched on.
rectangle at (700,395)-(736,431): text "%s"; shows DALI_Config.bBlinkzeit; tooltip Enter blink time (3 - 255 seconds); editable
rectangle at (40,80)-(761,474): text "Please wait!"; invisible if NOT DALI_Config.Unsichtbar
67 more shapes without text or variables
*)

(* Visualisation GroupSceneConfiguration
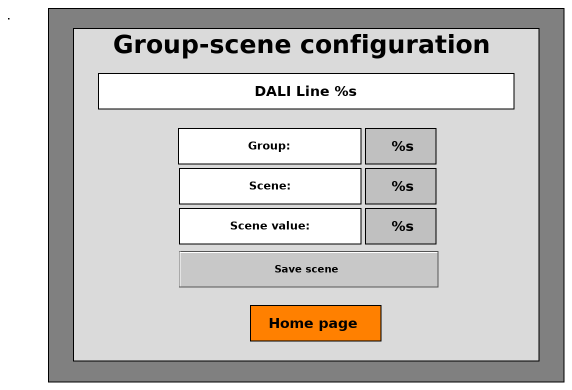
rectangle at (150,40)-(616,373): text "Group-scene configuration"
rounded rectangle at (327,317)-(458,353): text "Home page"; opens DALI; tooltip Back to home page
rounded rectangle at (175,85)-(591,121): text "DALI Line %s"; shows DALI_Config.bDali_Linie; tooltip You can change the DALI Line only on the home page.
rectangle at (255,140)-(438,176): text "Group:"
rectangle at (442,140)-(513,176): text "%s"; shows DALI_Config.sGroup; tooltip Enter the number of the group (1 - 16); editable
button at (256,263)-(515,299): text "Save scene"; taps DALI_Config.sSaveScene; tooltip Save the configured dim levels in the ECGs.
rectangle at (256,180)-(438,216): text "Scene:"
rectangle at (442,180)-(513,216): text "%s"; shows DALI_Config.sScene; tooltip Select scene 1 - 16; editable
rectangle at (256,220)-(438,256): text "Scene value:"
rectangle at (442,220)-(513,256): text "%s"; shows DALI_Config.sSceneValue; tooltip Select scene 1 - 16; editable
2 more shapes without text or variables
*)

